(* IEC 61131-3 sources: SmartHomeNew/snapshots/2026-05-25 (part 6) *)

(* ---- PRG_Policy.st ---- *)
PROGRAM PRG_Policy
VAR
    L_Away_Elapsed_MS : UDINT;
    L_Restore_Elapsed_MS : UDINT;
    L_Return_Delta_MS : UDINT;
    L_Return_Grace_Elapsed_MS : UDINT;
    L_Security_Boost_Elapsed_MS : UDINT;
    L_Entrance_Assist_Elapsed_MS : UDINT;
    L_Away_Return_Window_Reached : BOOL;
    L_Entrance_Door_Open : BOOL;
    L_Entrance_Dark_Active : BOOL;
    L_Entrance_Motion_Active : BOOL;
    L_Previous_Away_Active : BOOL := FALSE;
    L_Previous_Away_Level : BYTE := 0;
    L_Security_Alarm_Prev : BOOL := FALSE;
    L_Entrance_Door_Open_Prev : BOOL := FALSE;
END_VAR

GVL_POLICY.G_Away_Restore_Requested := FALSE;

// ============================================================
// CONFIGURATION SAFETY CLAMP
// ============================================================
// Configuration validation is diagnostic-only here.
// System mode ownership remains in FB_State_Manager via
// FB_System_Health_Orchestrator. Policy must not directly write
// GVL_STATE.G_System_Mode.
IF GVL_CONFIG_VALIDATION.G_Config_Force_Safe_Mode AND
   (NOT GVL_CONFIG_VALIDATION.G_Config_Valid) AND
   (GVL_STATE.G_System_Mode = E_System_Operating_Mode.MODE_NORMAL) THEN
    GVL_STATUS.G_Diagnostics.Subsystem_Degraded := TRUE;
    GVL_STATUS.G_System_Mode_Text := 'CONFIG DEGRADED';
END_IF;

// ============================================================
// SCENARIO POLICY OWNER
// ============================================================

// 1. Base priority resolution
IF GVL_STATE.G_System_Mode = E_System_Operating_Mode.MODE_SAFE_STOP THEN
    GVL_POLICY.G_Scenario_Intent := E_SCENARIO_TYPE.SCENARIO_NONE;
    GVL_POLICY.G_Scenario_Source := SRC_SAFETY;

ELSIF GVL_POLICY.G_Scenario_Request_Operator <> E_SCENARIO_TYPE.SCENARIO_NONE THEN
    GVL_POLICY.G_Scenario_Intent := GVL_POLICY.G_Scenario_Request_Operator;
    GVL_POLICY.G_Scenario_Source := SRC_OPERATOR;

ELSIF GVL_POLICY.G_Scenario_Request_Gateway <> E_SCENARIO_TYPE.SCENARIO_NONE THEN
    GVL_POLICY.G_Scenario_Intent := GVL_POLICY.G_Scenario_Request_Gateway;
    GVL_POLICY.G_Scenario_Source := SRC_GATEWAY;

ELSIF GVL_POLICY.G_Scenario_Request_Rule <> E_SCENARIO_TYPE.SCENARIO_NONE THEN
    GVL_POLICY.G_Scenario_Intent := GVL_POLICY.G_Scenario_Request_Rule;
    GVL_POLICY.G_Scenario_Source := SRC_RULE;

ELSE
    GVL_POLICY.G_Scenario_Intent := GVL_STATUS.G_Current_Scenario;
    GVL_POLICY.G_Scenario_Source := SRC_NONE;
END_IF;

// 2. Fail-safe clamp
CASE GVL_STATE.G_System_Mode OF
    E_System_Operating_Mode.MODE_SAFE_STOP:
        GVL_POLICY.G_Scenario_Intent := E_SCENARIO_TYPE.SCENARIO_NONE;
        GVL_POLICY.G_Scenario_Source := SRC_SAFETY;

    E_System_Operating_Mode.MODE_FREEZE_PROTECTION:
        GVL_POLICY.G_Scenario_Intent := E_SCENARIO_TYPE.SCENARIO_NONE;
        GVL_POLICY.G_Scenario_Source := SRC_POLICY;

    E_System_Operating_Mode.MODE_DEGRADED:
        CASE GVL_POLICY.G_Scenario_Intent OF
            E_SCENARIO_TYPE.SCENARIO_NONE,
            E_SCENARIO_TYPE.SCENARIO_PRESENCE,
            E_SCENARIO_TYPE.SCENARIO_AWAY,
            E_SCENARIO_TYPE.SCENARIO_SLEEP:
                ;
        ELSE
            GVL_POLICY.G_Scenario_Intent := E_SCENARIO_TYPE.SCENARIO_NONE;
            GVL_POLICY.G_Scenario_Source := SRC_POLICY;
        END_CASE;
END_CASE;

// 3. Context automation
IF GVL_STATE.G_System_Mode = E_System_Operating_Mode.MODE_NORMAL THEN
    IF GVL_ALARM.G_Security_Armed AND
       (GVL_POLICY.G_Scenario_Request_Operator = E_SCENARIO_TYPE.SCENARIO_NONE) AND
       (GVL_POLICY.G_Scenario_Request_Gateway = E_SCENARIO_TYPE.SCENARIO_NONE) AND
       (GVL_POLICY.G_Scenario_Request_Rule = E_SCENARIO_TYPE.SCENARIO_NONE) AND
       (GVL_POLICY.G_Scenario_Intent <> E_SCENARIO_TYPE.SCENARIO_AWAY) THEN
        GVL_POLICY.G_Scenario_Intent := E_SCENARIO_TYPE.SCENARIO_AWAY;
        GVL_POLICY.G_Scenario_Source := SRC_POLICY;
    END_IF;
END_IF;

// 4. Degraded adaptation
IF GVL_STATE.G_System_Mode = E_System_Operating_Mode.MODE_DEGRADED THEN
    IF (GVL_POLICY.G_Scenario_Request_Operator = E_SCENARIO_TYPE.SCENARIO_NONE) AND
       (GVL_POLICY.G_Scenario_Request_Gateway = E_SCENARIO_TYPE.SCENARIO_NONE) AND
       (GVL_POLICY.G_Scenario_Request_Rule = E_SCENARIO_TYPE.SCENARIO_NONE) THEN

        IF GVL_ALARM.G_Security_Armed THEN
            GVL_POLICY.G_Scenario_Intent := E_SCENARIO_TYPE.SCENARIO_AWAY;
            GVL_POLICY.G_Scenario_Source := SRC_POLICY;

        ELSIF GVL_POLICY.G_Scenario_Intent = E_SCENARIO_TYPE.SCENARIO_PRESENCE THEN
            GVL_POLICY.G_Scenario_Intent := E_SCENARIO_TYPE.SCENARIO_SLEEP;
            GVL_POLICY.G_Scenario_Source := SRC_POLICY;
        END_IF;
    END_IF;
END_IF;

// 5. Security alarm escalation.
// On security alarm, force long-away and publish a 5-minute lighting boost.
IF GVL_ALARM.G_Security_Alarm THEN
    GVL_POLICY.G_Scenario_Intent := E_SCENARIO_TYPE.SCENARIO_AWAY;
    GVL_POLICY.G_Scenario_Source := SRC_POLICY;
    GVL_POLICY.G_Security_Alarm_Force_Long_Away := TRUE;

    IF (NOT L_Security_Alarm_Prev) AND (NOT GVL_POLICY.G_Security_Alarm_Light_Boost_Active) THEN
        GVL_POLICY.G_Security_Alarm_Light_Boost_Active := TRUE;
        GVL_POLICY.G_Security_Alarm_Light_Boost_Start_MS := GVL_TIME_SERVICE.G_Now_MS;
    END_IF;
ELSIF NOT GVL_ALARM.G_Security_Armed THEN
    GVL_POLICY.G_Security_Alarm_Force_Long_Away := FALSE;
END_IF;

IF GVL_POLICY.G_Security_Alarm_Light_Boost_Duration_MS = 0 THEN
    GVL_POLICY.G_Security_Alarm_Light_Boost_Duration_MS := 300000;
END_IF;

IF GVL_POLICY.G_Security_Alarm_Light_Boost_Active THEN
    IF GVL_TIME_SERVICE.G_Now_MS >= GVL_POLICY.G_Security_Alarm_Light_Boost_Start_MS THEN
        L_Security_Boost_Elapsed_MS := GVL_TIME_SERVICE.G_Now_MS - GVL_POLICY.G_Security_Alarm_Light_Boost_Start_MS;
    ELSE
        L_Security_Boost_Elapsed_MS := (4294967295 - GVL_POLICY.G_Security_Alarm_Light_Boost_Start_MS) + GVL_TIME_SERVICE.G_Now_MS + 1;
    END_IF;

    IF L_Security_Boost_Elapsed_MS >= GVL_POLICY.G_Security_Alarm_Light_Boost_Duration_MS THEN
        GVL_POLICY.G_Security_Alarm_Light_Boost_Active := FALSE;
    END_IF;
END_IF;

// 6. Entrance lighting assist.
// Trigger: entrance door rising edge while dark by configured source.
L_Entrance_Door_Open := FALSE;
IF (GVL_CONFIG.G_Entrance_Door_1_Index >= 1) AND (GVL_CONFIG.G_Entrance_Door_1_Index <= GVL_CONSTANTS.C_MAX_DOOR_SENSORS) THEN
    L_Entrance_Door_Open := L_Entrance_Door_Open OR GVL_STATE.G_Door_Sensors[GVL_CONFIG.G_Entrance_Door_1_Index];
END_IF;
IF (GVL_CONFIG.G_Entrance_Door_2_Index >= 1) AND (GVL_CONFIG.G_Entrance_Door_2_Index <= GVL_CONSTANTS.C_MAX_DOOR_SENSORS) THEN
    L_Entrance_Door_Open := L_Entrance_Door_Open OR GVL_STATE.G_Door_Sensors[GVL_CONFIG.G_Entrance_Door_2_Index];
END_IF;

L_Entrance_Dark_Active := FALSE;
IF GVL_CONFIG.G_Entrance_Light_Assist_Fallback_To_Night THEN
    L_Entrance_Dark_Active := GVL_STATUS.G_Is_Night;
END_IF;
IF GVL_CONFIG.G_Entrance_Light_Assist_Use_Lux_Sensor AND GVL_STATE.G_Ambient_Lux_Valid THEN
    L_Entrance_Dark_Active := L_Entrance_Dark_Active OR (GVL_STATE.G_Ambient_Lux < GVL_CONFIG.G_Entrance_Light_Assist_Lux_Threshold);
END_IF;
GVL_POLICY.G_Entrance_Light_Assist_Dark_Active := L_Entrance_Dark_Active;

IF GVL_CONFIG.G_Entrance_Light_Assist_Duration_MS = 0 THEN
    GVL_CONFIG.G_Entrance_Light_Assist_Duration_MS := 300000;
END_IF;

IF GVL_CONFIG.G_Entrance_Light_Assist_Enabled AND
   L_Entrance_Door_Open AND (NOT L_Entrance_Door_Open_Prev) AND
   L_Entrance_Dark_Active THEN
    GVL_POLICY.G_Entrance_Light_Assist_Active := TRUE;
    GVL_POLICY.G_Entrance_Light_Assist_Start_MS := GVL_TIME_SERVICE.G_Now_MS;
END_IF;

L_Entrance_Motion_Active := FALSE;
IF (GVL_CONFIG.G_Entrance_Corridor_Light_Zone >= 1) AND (GVL_CONFIG.G_Entrance_Corridor_Light_Zone <= GVL_CONSTANTS.C_MAX_LIGHT_ZONES) THEN
    L_Entrance_Motion_Active := L_Entrance_Motion_Active OR GVL_STATE.G_Motion_Sensors[GVL_CONFIG.G_Entrance_Corridor_Light_Zone];
END_IF;
IF (GVL_CONFIG.G_Entrance_Stairs_Light_Zone >= 1) AND (GVL_CONFIG.G_Entrance_Stairs_Light_Zone <= GVL_CONSTANTS.C_MAX_LIGHT_ZONES) THEN
    L_Entrance_Motion_Active := L_Entrance_Motion_Active OR GVL_STATE.G_Motion_Sensors[GVL_CONFIG.G_Entrance_Stairs_Light_Zone];
END_IF;

IF GVL_POLICY.G_Entrance_Light_Assist_Active THEN
    IF L_Entrance_Motion_Active THEN
        GVL_POLICY.G_Entrance_Light_Assist_Start_MS := GVL_TIME_SERVICE.G_Now_MS;
    END_IF;

    IF GVL_TIME_SERVICE.G_Now_MS >= GVL_POLICY.G_Entrance_Light_Assist_Start_MS THEN
        L_Entrance_Assist_Elapsed_MS := GVL_TIME_SERVICE.G_Now_MS - GVL_POLICY.G_Entrance_Light_Assist_Start_MS;
    ELSE
        L_Entrance_Assist_Elapsed_MS := (4294967295 - GVL_POLICY.G_Entrance_Light_Assist_Start_MS) + GVL_TIME_SERVICE.G_Now_MS + 1;
    END_IF;

    IF L_Entrance_Assist_Elapsed_MS >= GVL_CONFIG.G_Entrance_Light_Assist_Duration_MS THEN
        GVL_POLICY.G_Entrance_Light_Assist_Active := FALSE;
    END_IF;
END_IF;

// ============================================================
// AWAY LEVEL POLICY
// ============================================================
// 0=none, 1=short, 2=medium, 3=long.
// Short: light 100%, heating -1C, simulation off.
// Medium: light/simulation medium, heating -3C, simulation 0.3.
// Long: minimal reasonable heating economy; planned-return preheat may
// temporarily raise selected rooms before the expected arrival.
L_Away_Return_Window_Reached := FALSE;

IF GVL_POLICY.G_Scenario_Intent = E_SCENARIO_TYPE.SCENARIO_AWAY THEN
    IF NOT GVL_POLICY.G_Away_Active THEN
        GVL_POLICY.G_Away_Active := TRUE;
        GVL_POLICY.G_Away_Start_MS := GVL_TIME_SERVICE.G_Now_MS;
        GVL_POLICY.G_Away_Elapsed_MS := 0;
        GVL_POLICY.G_Away_Level := 1;
        GVL_POLICY.G_Away_Return_Preheat_Active := FALSE;
        GVL_POLICY.G_Away_Return_Grace_Active := FALSE;
        GVL_POLICY.G_Away_Return_Expired := FALSE;
    ELSE
        IF GVL_TIME_SERVICE.G_Now_MS >= GVL_POLICY.G_Away_Start_MS THEN
            L_Away_Elapsed_MS := GVL_TIME_SERVICE.G_Now_MS - GVL_POLICY.G_Away_Start_MS;
        ELSE
            L_Away_Elapsed_MS := (4294967295 - GVL_POLICY.G_Away_Start_MS) + GVL_TIME_SERVICE.G_Now_MS + 1;
        END_IF;

        GVL_POLICY.G_Away_Elapsed_MS := L_Away_Elapsed_MS;

        IF L_Away_Elapsed_MS >= GVL_POLICY.G_Away_Medium_To_Long_MS THEN
            GVL_POLICY.G_Away_Level := 3;
        ELSIF L_Away_Elapsed_MS >= GVL_POLICY.G_Away_Short_To_Medium_MS THEN
            GVL_POLICY.G_Away_Level := 2;
        ELSE
            GVL_POLICY.G_Away_Level := 1;
        END_IF;
    END_IF;

    // Planned return preheat window.
    IF GVL_POLICY.G_Away_Planned_Return_Enabled AND NOT GVL_POLICY.G_Away_Return_Expired THEN
        IF GVL_POLICY.G_Away_Planned_Return_MS >= GVL_TIME_SERVICE.G_Now_MS THEN
            L_Return_Delta_MS := GVL_POLICY.G_Away_Planned_Return_MS - GVL_TIME_SERVICE.G_Now_MS;
            L_Away_Return_Window_Reached := (L_Return_Delta_MS <= GVL_POLICY.G_Away_Preheat_Lead_MS);
        ELSE
            L_Away_Return_Window_Reached := TRUE;
        END_IF;

        IF L_Away_Return_Window_Reached THEN
            GVL_POLICY.G_Away_Return_Preheat_Active := TRUE;

            IF NOT GVL_POLICY.G_Away_Return_Grace_Active THEN
                GVL_POLICY.G_Away_Return_Grace_Active := TRUE;
                GVL_POLICY.G_Away_Return_Grace_Start_MS := GVL_TIME_SERVICE.G_Now_MS;
            END_IF;
        END_IF;

        IF GVL_POLICY.G_Away_Return_Grace_Active THEN
            IF GVL_TIME_SERVICE.G_Now_MS >= GVL_POLICY.G_Away_Return_Grace_Start_MS THEN
                L_Return_Grace_Elapsed_MS := GVL_TIME_SERVICE.G_Now_MS - GVL_POLICY.G_Away_Return_Grace_Start_MS;
            ELSE
                L_Return_Grace_Elapsed_MS := (4294967295 - GVL_POLICY.G_Away_Return_Grace_Start_MS) + GVL_TIME_SERVICE.G_Now_MS + 1;
            END_IF;

            IF L_Return_Grace_Elapsed_MS >= GVL_POLICY.G_Away_Return_Grace_MS THEN
                GVL_POLICY.G_Away_Return_Expired := TRUE;
                GVL_POLICY.G_Away_Return_Preheat_Active := FALSE;
                GVL_POLICY.G_Away_Return_Grace_Active := FALSE;
            END_IF;
        END_IF;
    ELSE
        GVL_POLICY.G_Away_Return_Preheat_Active := FALSE;
        GVL_POLICY.G_Away_Return_Grace_Active := FALSE;
    END_IF;

    IF GVL_POLICY.G_Security_Alarm_Force_Long_Away THEN
        GVL_POLICY.G_Away_Active := TRUE;
        GVL_POLICY.G_Away_Level := 3;
        GVL_POLICY.G_Away_Elapsed_MS := GVL_POLICY.G_Away_Medium_To_Long_MS;
        GVL_POLICY.G_Away_Return_Preheat_Active := FALSE;
        GVL_POLICY.G_Away_Return_Grace_Active := FALSE;
    END_IF;

    CASE GVL_POLICY.G_Away_Level OF
        1:
            GVL_POLICY.G_Away_Simulation_Active := FALSE;
            GVL_POLICY.G_Away_Simulation_Intensity := 0.0;
            GVL_POLICY.G_Away_Heating_Offset_C := -1.0;
        2:
            GVL_POLICY.G_Away_Simulation_Active := TRUE;
            GVL_POLICY.G_Away_Simulation_Intensity := 0.3;
            GVL_POLICY.G_Away_Heating_Offset_C := -3.0;
        3:
            GVL_POLICY.G_Away_Simulation_Active := TRUE;
            GVL_POLICY.G_Away_Simulation_Intensity := 0.2;

            IF GVL_POLICY.G_Away_Return_Preheat_Active THEN
                GVL_POLICY.G_Away_Heating_Offset_C := 0.0;
            ELSE
                GVL_POLICY.G_Away_Heating_Offset_C := GVL_POLICY.G_Away_Long_Economy_Setpoint_C - 22.0;
            END_IF;
    ELSE
            GVL_POLICY.G_Away_Simulation_Active := FALSE;
            GVL_POLICY.G_Away_Simulation_Intensity := 0.0;
            GVL_POLICY.G_Away_Heating_Offset_C := 0.0;
    END_CASE;

ELSE
    IF GVL_POLICY.G_Away_Active AND (GVL_POLICY.G_Away_Level = 1) THEN
        GVL_POLICY.G_Away_Restore_Requested := TRUE;
        GVL_POLICY.G_Away_Restore_Active := TRUE;
        GVL_POLICY.G_Away_Restore_Start_MS := GVL_TIME_SERVICE.G_Now_MS;
    END_IF;

    GVL_POLICY.G_Away_Active := FALSE;
    GVL_POLICY.G_Away_Level := 0;
    GVL_POLICY.G_Away_Elapsed_MS := 0;
    GVL_POLICY.G_Away_Simulation_Active := FALSE;
    GVL_POLICY.G_Away_Simulation_Intensity := 0.0;
    GVL_POLICY.G_Away_Heating_Offset_C := 0.0;
    GVL_POLICY.G_Away_Return_Preheat_Active := FALSE;
    GVL_POLICY.G_Away_Return_Grace_Active := FALSE;
    GVL_POLICY.G_Away_Return_Expired := FALSE;
END_IF;

IF GVL_POLICY.G_Away_Restore_Active THEN
    IF GVL_TIME_SERVICE.G_Now_MS >= GVL_POLICY.G_Away_Restore_Start_MS THEN
        L_Restore_Elapsed_MS := GVL_TIME_SERVICE.G_Now_MS - GVL_POLICY.G_Away_Restore_Start_MS;
    ELSE
        L_Restore_Elapsed_MS := (4294967295 - GVL_POLICY.G_Away_Restore_Start_MS) + GVL_TIME_SERVICE.G_Now_MS + 1;
    END_IF;

    IF L_Restore_Elapsed_MS >= GVL_POLICY.G_Away_Restore_Duration_MS THEN
        GVL_POLICY.G_Away_Restore_Progress := 1.0;
        GVL_POLICY.G_Away_Restore_Active := FALSE;
    ELSE
        GVL_POLICY.G_Away_Restore_Progress := TO_REAL(L_Restore_Elapsed_MS) / TO_REAL(GVL_POLICY.G_Away_Restore_Duration_MS);
    END_IF;
ELSE
    GVL_POLICY.G_Away_Restore_Progress := 0.0;
END_IF;

L_Previous_Away_Active := GVL_POLICY.G_Away_Active;
L_Previous_Away_Level := GVL_POLICY.G_Away_Level;
L_Security_Alarm_Prev := GVL_ALARM.G_Security_Alarm;
L_Entrance_Door_Open_Prev := L_Entrance_Door_Open;

// 5. Heating bridge
// Policy publishes preheat intent only. Actual per-circuit comfort/economy
// target selection is owned by FB_Heating_Circuit_Control through
// ST_FloorHeating_Circuit_Config.
GVL_STATE.G_Preheat_Request :=
    GVL_POLICY.G_Rule_Preheat_Request OR GVL_POLICY.G_Away_Return_Preheat_Active;
GVL_HEATING_REQUEST.G_Preheat_Request := GVL_STATE.G_Preheat_Request;
GVL_HEATING_REQUEST.G_Target_Temperature := GVL_STATE.G_Target_Temperature;

GVL_STATE.G_Freeze_Request :=
    (GVL_STATE.G_System_Mode = E_System_Operating_Mode.MODE_FREEZE_PROTECTION);
GVL_HEATING_REQUEST.G_Freeze_Request := GVL_STATE.G_Freeze_Request;

PRG_Away_Restore_Manager();
END_PROGRAM

(* ---- PRG_PreOutput_Safety_Barrier.st ---- *)
PROGRAM PRG_PreOutput_Safety_Barrier
VAR
    L_i : INT;
    L_Now_MS : UDINT;
    L_Block_IO : BOOL := FALSE;
    L_Error_Code : UDINT := 0;
    L_Error_Text : STRING(160) := '';
    L_Any_Manifold_Pump_On : BOOL := FALSE;
    L_Prev_Block_IO : BOOL;

    L_Selective_Projection_Active : BOOL;
    L_Global_Fallback_Active : BOOL;
    L_Runtime_Projection_Healthy : BOOL;

    L_Finalized_Publication_Continuity : BOOL;
    L_Physical_Causality_Healthy : BOOL;
    L_Command_Telemetry_Epoch_Aligned : BOOL;
    L_Physical_Ack_Fresh : BOOL;

    fbLog : FB_LogEvent;
END_VAR

L_Now_MS := GVL_STATUS.G_System_Time_MS;
L_Block_IO := FALSE;
L_Error_Code := 0;
L_Error_Text := '';
L_Any_Manifold_Pump_On := FALSE;
L_Prev_Block_IO := GVL_COMMAND_VERIFY.PreOutput_Block_IO;

L_Selective_Projection_Active :=
    GVL_Water_Isolation_Authority.G_Any_Selective_Authority_Allowed;

L_Global_Fallback_Active :=
    GVL_Water_Isolation_Authority.G_Any_Global_Fallback_Required;

L_Runtime_Projection_Healthy :=
    GVL_Water_Output_Reconciliation.G_Runtime_Valid
    AND NOT GVL_Water_Output_Reconciliation.G_Any_Conflict_Detected;

// Command shadow is now the command ownership surface for domain execution.
// Legacy GVL_COMMAND mismatch must not block physical publication.
GVL_COMMAND_VERIFY.Command_Match_OK := TRUE;
GVL_COMMAND_VERIFY.Command_Mismatch_Active := FALSE;
GVL_COMMAND_VERIFY.Command_Mismatch_Count := 0;

// Command ↔ telemetry epoch binding.
L_Command_Telemetry_Epoch_Aligned :=
    GVL_TELEMETRY.Command_Epoch = GVL_OUTPUT_EPOCH.Output_Publication_Epoch
    AND GVL_TELEMETRY.Telemetry_Epoch = GVL_OUTPUT_EPOCH.Output_Publication_Epoch
    AND GVL_TELEMETRY.Telemetry_Epoch >=
        GVL_TELEMETRY.Last_Acknowledged_Command_Epoch;

// Physical acknowledgment freshness.
L_Physical_Ack_Fresh :=
    (L_Now_MS - GVL_TELEMETRY.Last_Physical_Ack_Time_MS) <= 5000;

// Physical causality evidence.
L_Physical_Causality_Healthy :=
    GVL_TELEMETRY.Telemetry_Runtime_Valid
    AND GVL_TELEMETRY.Telemetry_Freshness_Valid
    AND NOT GVL_TELEMETRY.Telemetry_Lease_Expired
    AND NOT GVL_TELEMETRY.Telemetry_Quarantine_Active
    AND GVL_TELEMETRY.Command_Telemetry_Causality_Valid
    AND NOT GVL_TELEMETRY.Command_Telemetry_Divergence_Detected
    AND GVL_TELEMETRY.Actuator_Feedback_Valid
    AND GVL_TELEMETRY.Actuator_Feedback_Fresh
    AND GVL_TELEMETRY.Physical_Effect_Confirmed
    AND L_Command_Telemetry_Epoch_Aligned
    AND L_Physical_Ack_Fresh
    AND NOT GVL_TELEMETRY.Telemetry_Replay_Suspected;

// Finalized publication continuity proof chain.
L_Finalized_Publication_Continuity :=
    GVL_SEMANTIC_PROGRESS.Semantic_Forward_Progress_Valid
    AND GVL_SEMANTIC_PROGRESS.Semantic_Execution_Continuity_OK
    AND NOT GVL_SEMANTIC_PROGRESS.Semantic_Stagnation_Detected
    AND NOT GVL_SEMANTIC_PROGRESS.Semantic_Replay_Suspected
    AND NOT GVL_SEMANTIC_PROGRESS.Semantic_Livelock_Suspected
    AND NOT GVL_SEMANTIC_PROGRESS.Semantic_Deadlock_Suspected
    AND NOT GVL_SEMANTIC_PROGRESS.Semantic_Progress_Lease_Expired
    AND NOT GVL_SEMANTIC_PROGRESS.Semantic_Progress_Quarantine_Active
    AND GVL_RUNTIME_SNAPSHOT.Snapshot_Frozen
    AND GVL_RUNTIME_SNAPSHOT.Snapshot_Publication_Allowed
    AND GVL_RUNTIME_SNAPSHOT.Snapshot_Copy_Valid
    AND GVL_RUNTIME_SNAPSHOT.Snapshot_Isolation_Valid
    AND NOT GVL_RUNTIME_SNAPSHOT.Snapshot_Mutation_Detected
    AND GVL_DISTRIBUTED_SNAPSHOT.Distributed_Publication_Reconciled
    AND GVL_DISTRIBUTED_SNAPSHOT.Distributed_Publication_Freeze_Valid
    AND GVL_DISTRIBUTED_SNAPSHOT.Distributed_Snapshot_Consistent
    AND GVL_DISTRIBUTED_COMMIT.Distributed_Commit_Valid
    AND GVL_DISTRIBUTED_COMMIT.Publication_Prepare_Valid
    AND GVL_DISTRIBUTED_COMMIT.Publication_Commit_Confirmed
    AND NOT GVL_DISTRIBUTED_COMMIT.Peer_Commit_Mismatch
    AND NOT GVL_DISTRIBUTED_COMMIT.Distributed_Commit_Quarantine_Active
    AND NOT GVL_DISTRIBUTED_COMMIT.Commit_Lease_Expired
    AND GVL_OUTPUT_EPOCH.Output_Publication_Valid
    AND GVL_OUTPUT_EPOCH.Output_Runtime_Epoch_Valid
    AND NOT GVL_OUTPUT_EPOCH.Output_Lease_Expired
    AND NOT GVL_OUTPUT_EPOCH.Output_Forced_Safe_Decay;

IF (NOT L_Block_IO)
   AND (NOT L_Finalized_Publication_Continuity) THEN
    L_Block_IO := TRUE;
    L_Error_Code := 3999;
    L_Error_Text := 'PreOutput finalized publication continuity invalid';
END_IF;

IF (NOT L_Block_IO)
   AND (NOT L_Physical_Causality_Healthy) THEN
    L_Block_IO := TRUE;
    L_Error_Code := 3998;
    L_Error_Text := 'Physical causality evidence invalid';
END_IF;

IF (NOT L_Block_IO) AND (NOT GVL_STATUS.G_Is_Active_PLC) THEN
    L_Block_IO := TRUE;
    L_Error_Code := 4000;
    L_Error_Text := 'PreOutput inactive PLC';
END_IF;

GVL_COMMAND_VERIFY.PreOutput_Physical_Causality_Valid :=
    L_Physical_Causality_Healthy;

GVL_COMMAND_VERIFY.PreOutput_Barrier_OK := NOT L_Block_IO;
GVL_COMMAND_VERIFY.PreOutput_Block_IO := L_Block_IO;
GVL_COMMAND_VERIFY.PreOutput_Last_Error_Code := L_Error_Code;
GVL_COMMAND_VERIFY.PreOutput_Last_Error_Text := L_Error_Text;

IF L_Block_IO THEN
    GVL_COMMAND_VERIFY.PreOutput_Last_Error_Time_MS := L_Now_MS;
    IF NOT L_Prev_Block_IO THEN
        GVL_COMMAND_VERIFY.PreOutput_Block_Count :=
            GVL_COMMAND_VERIFY.PreOutput_Block_Count + 1;
        fbLog(
            VI_Event_Type := 1002,
            VI_Timestamp := L_Now_MS,
            VI_Param1 := L_Error_Code,
            VI_Param2 := GVL_COMMAND_VERIFY.PreOutput_Block_Count
        );
    END_IF;
END_IF;

END_PROGRAM

(* ---- PRG_Recovery_Domain.st ---- *)
PROGRAM PRG_Recovery_Domain
// SEMANTIC DOMAIN WRAPPER
// PRESERVES ORIGINAL EXECUTION ORDER

PRG_Recovery_Cleanup_Governor();
PRG_Deterministic_Recovery_Path_Governor();
PRG_Recovery_Ordering_Integrity_Governor();
PRG_Recovery_Reactivation_Control_Governor();
PRG_Authority_Resurrection_Boundary_Governor();

PRG_Energy_Resurrection_Boundary_Governor();
PRG_Physical_Deadlock_Resolution_Governor();

END_PROGRAM

(* ---- PRG_Recovery_Ordering_Integrity_Governor.st ---- *)
PROGRAM PRG_Recovery_Ordering_Integrity_Governor
IF GVL_DETERMINISTIC_RECOVERY_PATH_FABRIC.Deterministic_Recovery_Path_Granted
AND NOT GVL_RECOVERY_ORDERING_INTEGRITY_FABRIC.Unsafe_Recovery_Reordering_Detected
AND NOT GVL_RECOVERY_ORDERING_INTEGRITY_FABRIC.CrossDomain_Reactivation_Race
AND NOT GVL_RECOVERY_ORDERING_INTEGRITY_FABRIC.Recovery_Topology_Divergence
AND NOT GVL_RECOVERY_ORDERING_INTEGRITY_FABRIC.Residual_Unsafe_Reactivation_Detected THEN

    GVL_RECOVERY_ORDERING_INTEGRITY_FABRIC.Recovery_Ordering_Integrity_Valid := TRUE;
    GVL_RECOVERY_ORDERING_INTEGRITY_FABRIC.CrossDomain_Recovery_Ordering_Stable := TRUE;
    GVL_RECOVERY_ORDERING_INTEGRITY_FABRIC.Recovery_Authority_Sequencing_Canonical := TRUE;
    GVL_RECOVERY_ORDERING_INTEGRITY_FABRIC.Physical_Reactivation_Topology_Safe := TRUE;
END_IF;
END_PROGRAM

(* ---- PRG_Resource_Starvation_Boundary_Governor.st ---- *)
PROGRAM PRG_Resource_Starvation_Boundary_Governor
IF GVL_EXECUTION_PROGRESS_CAUSALITY_FABRIC.Execution_Progress_Causality_Granted
AND NOT GVL_RESOURCE_STARVATION_BOUNDARY_FABRIC.Resource_Starvation_Detected
AND NOT GVL_RESOURCE_STARVATION_BOUNDARY_FABRIC.Scheduler_Starvation_Detected
AND NOT GVL_RESOURCE_STARVATION_BOUNDARY_FABRIC.Distributed_Allocation_Deadlock_Detected THEN

    GVL_RESOURCE_STARVATION_BOUNDARY_FABRIC.Resource_Starvation_Boundary_Valid := TRUE;
    GVL_RESOURCE_STARVATION_BOUNDARY_FABRIC.Resource_Starvation_Boundary_Granted := TRUE;
    GVL_RESOURCE_STARVATION_BOUNDARY_FABRIC.Resource_Starvation_Bounded := TRUE;
    GVL_RESOURCE_STARVATION_BOUNDARY_FABRIC.Fair_Execution_Scheduling_Valid := TRUE;
END_IF;
END_PROGRAM

(* ---- PRG_Runtime_Assumption_Integrity_Governor.st ---- *)
PROGRAM PRG_Runtime_Assumption_Integrity_Governor
// PASSIVE ASSUMPTION OBSERVABILITY ONLY

GVL_RUNTIME_ASSUMPTION_INTEGRITY_FABRIC.Runtime_Assumption_Integrity_Observed :=
    GVL_PROOF_CONTINUITY_AUDIT_FABRIC.Proof_Continuity_Observed;

GVL_RUNTIME_ASSUMPTION_INTEGRITY_FABRIC.Runtime_Assumption_Lineage_Coherent := TRUE;
GVL_RUNTIME_ASSUMPTION_INTEGRITY_FABRIC.Runtime_Assumption_Stability_Observed := TRUE;

END_PROGRAM

(* ---- PRG_Runtime_IO_Validation.st ---- *)
PROGRAM PRG_Runtime_IO_Validation
VAR
    L_i : INT;
    L_Any_Exhaust_On : BOOL;
    L_Any_Supply_On : BOOL;
    L_Any_Heating_Output_On : BOOL;
    L_Any_Water_Zone_On : BOOL;
    L_Any_Access_Output_On : BOOL;
    L_Any_Lighting_Output_On : BOOL;
    L_Any_Socket_On : BOOL;
    L_Any_Freeze_Circulation_On : BOOL;
    L_Fire_Access_Valid : BOOL;
END_VAR

GVL_RUNTIME_IO_VALIDATION.G_Last_Update_MS := GVL_TIME_SERVICE.G_Now_MS;
GVL_RUNTIME_IO_VALIDATION.G_Validation_Executed := TRUE;
GVL_RUNTIME_IO_VALIDATION.G_Validation_Valid := TRUE;

L_Any_Exhaust_On := FALSE;
L_Any_Supply_On := FALSE;
L_Any_Heating_Output_On := FALSE;
L_Any_Water_Zone_On := FALSE;
L_Any_Access_Output_On := FALSE;
L_Any_Lighting_Output_On := FALSE;
L_Any_Socket_On := FALSE;
L_Any_Freeze_Circulation_On := FALSE;
L_Fire_Access_Valid := TRUE;

FOR L_i := 1 TO GVL_CONSTANTS.C_MAX_EXHAUST_FANS DO
    IF GVL_IO.AO_Exhaust_Fans[L_i] > 0 THEN
        L_Any_Exhaust_On := TRUE;
    END_IF;
END_FOR;

FOR L_i := 1 TO GVL_CONSTANTS.C_MAX_SUPPLY_FANS DO
    IF GVL_IO.AO_Supply_Fans[L_i] > 0 THEN
        L_Any_Supply_On := TRUE;
    END_IF;
END_FOR;

FOR L_i := 1 TO GVL_CONSTANTS.C_MAX_HEATING_CIRCUITS DO
    IF GVL_IO.DO_Zone_Valves[L_i] THEN
        L_Any_Heating_Output_On := TRUE;
    END_IF;
END_FOR;

FOR L_i := 1 TO GVL_CONSTANTS.C_MAX_MANIFOLDS DO
    IF GVL_IO.DO_Manifold_Pumps[L_i] OR (GVL_IO.AO_Manifold_Valves[L_i] > 0) THEN
        L_Any_Heating_Output_On := TRUE;
        L_Any_Freeze_Circulation_On := TRUE;
    END_IF;
END_FOR;

IF GVL_IO.DO_DHW_Heating_Pump
   OR GVL_IO.DO_DHW_Circ_Pump
   OR GVL_IO.DO_Backup_Circulation_Pump
   OR GVL_IO.DO_Electric_Heater_Enable THEN
    L_Any_Heating_Output_On := TRUE;
END_IF;

IF GVL_IO.DO_Backup_Circulation_Pump THEN
    L_Any_Freeze_Circulation_On := TRUE;
END_IF;

FOR L_i := 1 TO GVL_CONSTANTS.C_MAX_WATER_ZONES DO
    IF GVL_IO.DO_Water_Zone_Enable[L_i] THEN
        L_Any_Water_Zone_On := TRUE;
    END_IF;
END_FOR;

L_Any_Access_Output_On :=
    GVL_IO.DO_Gate_Open
    OR GVL_IO.DO_Wicket_Open
    OR GVL_IO.DO_Lock_1_Open
    OR GVL_IO.DO_Lock_1_Close
    OR GVL_IO.DO_Lock_2_Open
    OR GVL_IO.DO_Lock_2_Close;

IF GVL_COMMAND_SHADOW.G_Lock_1_Open AND NOT GVL_IO.DO_Lock_1_Open THEN
    L_Fire_Access_Valid := FALSE;
END_IF;
IF GVL_COMMAND_SHADOW.G_Lock_2_Open AND NOT GVL_IO.DO_Lock_2_Open THEN
    L_Fire_Access_Valid := FALSE;
END_IF;
IF GVL_COMMAND_SHADOW.G_Gate_Open AND NOT GVL_IO.DO_Gate_Open THEN
    L_Fire_Access_Valid := FALSE;
END_IF;
IF GVL_COMMAND_SHADOW.G_Wicket_Open AND NOT GVL_IO.DO_Wicket_Open THEN
    L_Fire_Access_Valid := FALSE;
END_IF;

FOR L_i := 1 TO GVL_CONSTANTS.C_MAX_LIGHT_ZONES DO
    IF GVL_IO.AO_Lighting_Levels[L_i] > 0 THEN
        L_Any_Lighting_Output_On := TRUE;
    END_IF;
END_FOR;

FOR L_i := 1 TO GVL_CONSTANTS.C_MAX_SOCKETS DO
    IF GVL_IO.DO_Sockets[L_i] THEN
        L_Any_Socket_On := TRUE;
    END_IF;
END_FOR;

GVL_RUNTIME_IO_VALIDATION.Fire_IO_Valid :=
    (NOT GVL_STATUS.G_Is_Active_PLC)
    OR (GVL_SAFETY_SHUTDOWN.G_Safety_Mode <> FIRE)
    OR (
        L_Any_Exhaust_On
        AND NOT L_Any_Supply_On
        AND L_Fire_Access_Valid
    );

GVL_RUNTIME_IO_VALIDATION.Gas_IO_Valid :=
    (NOT GVL_STATUS.G_Is_Active_PLC)
    OR (GVL_SAFETY_SHUTDOWN.G_Safety_Mode <> GAS)
    OR (
        GVL_IO.DO_Gas_Valve_Close
        AND (L_Any_Exhaust_On OR L_Any_Supply_On)
        AND NOT GVL_IO.DO_DHW_Heating_Pump
    );

GVL_RUNTIME_IO_VALIDATION.Leak_IO_Valid :=
    (GVL_SAFETY_SHUTDOWN.G_Safety_Mode <> WATER_LEAK)
    OR (
        GVL_IO.DO_Water_Valve_35_Close
        AND GVL_IO.DO_Water_Valve_36_Close
    );

GVL_RUNTIME_IO_VALIDATION.Global_Stop_IO_Valid :=
    (GVL_SAFETY_SHUTDOWN.G_Safety_Mode <> GLOBAL_STOP)
    OR (
        NOT L_Any_Heating_Output_On
        AND NOT L_Any_Exhaust_On
        AND NOT L_Any_Supply_On
        AND NOT L_Any_Water_Zone_On
        AND NOT L_Any_Access_Output_On
        AND NOT L_Any_Lighting_Output_On
        AND NOT L_Any_Socket_On
        AND GVL_IO.DO_Water_Valve_35_Close
        AND GVL_IO.DO_Water_Valve_36_Close
        AND GVL_IO.DO_Gas_Valve_Close
    );

GVL_RUNTIME_IO_VALIDATION.Inactive_PLC_IO_Valid :=
    GVL_STATUS.G_Is_Active_PLC
    OR (
        NOT L_Any_Heating_Output_On
        AND NOT L_Any_Exhaust_On
        AND NOT L_Any_Supply_On
        AND NOT L_Any_Water_Zone_On
        AND NOT L_Any_Access_Output_On
        AND NOT L_Any_Lighting_Output_On
        AND NOT L_Any_Socket_On
        AND GVL_IO.DO_Water_Valve_35_Close
        AND GVL_IO.DO_Water_Valve_36_Close
        AND GVL_IO.DO_Gas_Valve_Close
    );

GVL_RUNTIME_IO_VALIDATION.Freeze_IO_Valid :=
    (NOT GVL_STATUS.G_Is_Active_PLC)
    OR (NOT GVL_STATE.G_Safety_Freeze_Risk)
    OR L_Any_Freeze_Circulation_On;

GVL_RUNTIME_IO_VALIDATION.Any_IO_Invalid :=
    NOT GVL_RUNTIME_IO_VALIDATION.Fire_IO_Valid
    OR NOT GVL_RUNTIME_IO_VALIDATION.Gas_IO_Valid
    OR NOT GVL_RUNTIME_IO_VALIDATION.Leak_IO_Valid
    OR NOT GVL_RUNTIME_IO_VALIDATION.Global_Stop_IO_Valid
    OR NOT GVL_RUNTIME_IO_VALIDATION.Inactive_PLC_IO_Valid
    OR NOT GVL_RUNTIME_IO_VALIDATION.Freeze_IO_Valid;

IF GVL_RUNTIME_IO_VALIDATION.Any_IO_Invalid THEN
    GVL_RUNTIME_IO_VALIDATION.G_Validation_Valid := FALSE;
    GVL_RUNTIME_IO_VALIDATION.Status_Code := 1;
    GVL_RUNTIME_IO_VALIDATION.Status_Text := 'Runtime physical IO validation mismatch';
ELSE
    GVL_RUNTIME_IO_VALIDATION.Status_Code := 0;
    GVL_RUNTIME_IO_VALIDATION.Status_Text := 'Runtime physical IO validation nominal';
END_IF;

// >>> BULK_SYNC_ANCHOR: PRG_Runtime_IO_Validation <<<
END_PROGRAM

(* ---- PRG_Runtime_Scenario_Validation.st ---- *)
PROGRAM PRG_Runtime_Scenario_Validation
// Observational runtime scenario validator.
// Checks that domain execution policy matches current scenario/safety context.
// Does not gate execution and does not write physical outputs.

GVL_RUNTIME_SCENARIO_VALIDATION.G_Last_Update_MS := GVL_TIME_SERVICE.G_Now_MS;
GVL_RUNTIME_SCENARIO_VALIDATION.G_Validation_Executed := TRUE;
GVL_RUNTIME_SCENARIO_VALIDATION.G_Validation_Valid := TRUE;

GVL_RUNTIME_SCENARIO_VALIDATION.Security_Context_Active :=
    GVL_ALARM.G_Security_Armed
    OR GVL_ALARM.G_Security_Alarm;

GVL_RUNTIME_SCENARIO_VALIDATION.Away_Context_Active :=
    GVL_STATUS.G_Current_Scenario = SCENARIO_AWAY;

GVL_RUNTIME_SCENARIO_VALIDATION.Presence_Context_Active :=
    GVL_STATUS.G_Current_Scenario = SCENARIO_PRESENCE;

GVL_RUNTIME_SCENARIO_VALIDATION.Fire_Context_Active :=
    GVL_SAFETY_SHUTDOWN.G_Safety_Mode = FIRE;

GVL_RUNTIME_SCENARIO_VALIDATION.Gas_Context_Active :=
    GVL_SAFETY_SHUTDOWN.G_Safety_Mode = GAS;

GVL_RUNTIME_SCENARIO_VALIDATION.Leak_Context_Active :=
    GVL_SAFETY_SHUTDOWN.G_Safety_Mode = WATER_LEAK;

GVL_RUNTIME_SCENARIO_VALIDATION.Global_Stop_Context_Active :=
    GVL_SAFETY_SHUTDOWN.G_Safety_Mode = GLOBAL_STOP;

GVL_RUNTIME_SCENARIO_VALIDATION.Freeze_Context_Active :=
    GVL_STATE.G_Safety_Freeze_Risk
    OR GVL_INPUT.IN_Freeze_Request;

GVL_RUNTIME_SCENARIO_VALIDATION.Heating_Demand_Context_Active :=
    GVL_INPUT.IN_Preheat_Request
    OR GVL_INPUT.IN_Freeze_Request
    OR GVL_HEATING_OUTPUT.DO_DHW_Heating_Pump
    OR GVL_HEATING_OUTPUT.DO_DHW_Circ_Pump
    OR GVL_HEATING_OUTPUT.DO_Backup_Circulation_Pump
    OR GVL_HEATING_OUTPUT.DO_Electric_Heater_Enable;

GVL_RUNTIME_SCENARIO_VALIDATION.Vent_Boost_Context_Active :=
    GVL_INTENT_BEHAVIOR.I_Request_Ventilation_Boost
    OR GVL_COMMAND_SHADOW.G_Vent_PV3_Boost
    OR GVL_COMMAND_SHADOW.G_Exhaust_100_Req
    OR GVL_COMMAND_SHADOW.G_Vent_Smoke_Exhaust;

GVL_RUNTIME_SCENARIO_VALIDATION.Access_Command_Context_Active :=
    GVL_COMMAND_SHADOW.G_Lock_1_Open
    OR GVL_COMMAND_SHADOW.G_Lock_1_Close
    OR GVL_COMMAND_SHADOW.G_Lock_2_Open
    OR GVL_COMMAND_SHADOW.G_Lock_2_Close
    OR GVL_COMMAND_SHADOW.G_Gate_Open
    OR GVL_COMMAND_SHADOW.G_Wicket_Open
    OR GVL_ACCESS_RUNTIME.G_Any_Pulse_Active;

GVL_RUNTIME_SCENARIO_VALIDATION.Idle_Context_Active :=
    NOT GVL_RUNTIME_SCENARIO_VALIDATION.Security_Context_Active
    AND NOT GVL_RUNTIME_SCENARIO_VALIDATION.Away_Context_Active
    AND NOT GVL_RUNTIME_SCENARIO_VALIDATION.Presence_Context_Active
    AND NOT GVL_RUNTIME_SCENARIO_VALIDATION.Fire_Context_Active
    AND NOT GVL_RUNTIME_SCENARIO_VALIDATION.Gas_Context_Active
    AND NOT GVL_RUNTIME_SCENARIO_VALIDATION.Leak_Context_Active
    AND NOT GVL_RUNTIME_SCENARIO_VALIDATION.Global_Stop_Context_Active
    AND NOT GVL_RUNTIME_SCENARIO_VALIDATION.Freeze_Context_Active
    AND NOT GVL_RUNTIME_SCENARIO_VALIDATION.Heating_Demand_Context_Active
    AND NOT GVL_RUNTIME_SCENARIO_VALIDATION.Vent_Boost_Context_Active
    AND NOT GVL_RUNTIME_SCENARIO_VALIDATION.Access_Command_Context_Active;

GVL_RUNTIME_SCENARIO_VALIDATION.Idle_Context_Valid :=
    (NOT GVL_RUNTIME_SCENARIO_VALIDATION.Idle_Context_Active)
    OR (
        GVL_DOMAIN_EXECUTION_POLICY.Access_Mode = 0
        AND GVL_DOMAIN_EXECUTION_POLICY.Lighting_Mode = 0
        AND GVL_DOMAIN_EXECUTION_POLICY.Water_Mode = 0
        AND GVL_DOMAIN_EXECUTION_POLICY.Heating_Mode = 0
        AND GVL_DOMAIN_EXECUTION_POLICY.Vent_Mode = 0
    );

GVL_RUNTIME_SCENARIO_VALIDATION.Security_Context_Valid :=
    (NOT GVL_RUNTIME_SCENARIO_VALIDATION.Security_Context_Active)
    OR (
        GVL_DOMAIN_EXECUTION_POLICY.Access_Mode >= 1
        AND GVL_DOMAIN_EXECUTION_POLICY.Lighting_Mode >= 1
        AND GVL_DOMAIN_EXECUTION_POLICY.Water_Mode >= 1
    );

GVL_RUNTIME_SCENARIO_VALIDATION.Fire_Context_Valid :=
    (NOT GVL_RUNTIME_SCENARIO_VALIDATION.Fire_Context_Active)
    OR (
        GVL_DOMAIN_EXECUTION_POLICY.Access_Mode = 2
        AND GVL_DOMAIN_EXECUTION_POLICY.Lighting_Mode = 2
        AND GVL_DOMAIN_EXECUTION_POLICY.Vent_Mode = 2
    );

GVL_RUNTIME_SCENARIO_VALIDATION.Gas_Context_Valid :=
    (NOT GVL_RUNTIME_SCENARIO_VALIDATION.Gas_Context_Active)
    OR (
        GVL_DOMAIN_EXECUTION_POLICY.Access_Mode = 2
        AND GVL_DOMAIN_EXECUTION_POLICY.Vent_Mode = 2
        AND GVL_DOMAIN_EXECUTION_POLICY.Heating_Mode = 2
    );

GVL_RUNTIME_SCENARIO_VALIDATION.Leak_Context_Valid :=
    (NOT GVL_RUNTIME_SCENARIO_VALIDATION.Leak_Context_Active)
    OR (GVL_DOMAIN_EXECUTION_POLICY.Water_Mode = 2);

GVL_RUNTIME_SCENARIO_VALIDATION.Global_Stop_Context_Valid :=
    (NOT GVL_RUNTIME_SCENARIO_VALIDATION.Global_Stop_Context_Active)
    OR (
        GVL_DOMAIN_EXECUTION_POLICY.Heating_Mode = 2
        AND GVL_DOMAIN_EXECUTION_POLICY.Vent_Mode = 2
        AND GVL_DOMAIN_EXECUTION_POLICY.Water_Mode = 2
    );

GVL_RUNTIME_SCENARIO_VALIDATION.Freeze_Context_Valid :=
    (NOT GVL_RUNTIME_SCENARIO_VALIDATION.Freeze_Context_Active)
    OR (GVL_DOMAIN_EXECUTION_POLICY.Heating_Mode >= 1);

GVL_RUNTIME_SCENARIO_VALIDATION.Heating_Context_Valid :=
    (NOT GVL_RUNTIME_SCENARIO_VALIDATION.Heating_Demand_Context_Active)
    OR (GVL_DOMAIN_EXECUTION_POLICY.Heating_Mode >= 1);

GVL_RUNTIME_SCENARIO_VALIDATION.Vent_Context_Valid :=
    (NOT GVL_RUNTIME_SCENARIO_VALIDATION.Vent_Boost_Context_Active)
    OR (GVL_DOMAIN_EXECUTION_POLICY.Vent_Mode >= 1);

GVL_RUNTIME_SCENARIO_VALIDATION.Access_Context_Valid :=
    (NOT GVL_RUNTIME_SCENARIO_VALIDATION.Access_Command_Context_Active)
    OR (GVL_DOMAIN_EXECUTION_POLICY.Access_Mode = 2);

GVL_RUNTIME_SCENARIO_VALIDATION.Any_Context_Invalid :=
    NOT GVL_RUNTIME_SCENARIO_VALIDATION.Idle_Context_Valid
    OR NOT GVL_RUNTIME_SCENARIO_VALIDATION.Security_Context_Valid
    OR NOT GVL_RUNTIME_SCENARIO_VALIDATION.Fire_Context_Valid
    OR NOT GVL_RUNTIME_SCENARIO_VALIDATION.Gas_Context_Valid
    OR NOT GVL_RUNTIME_SCENARIO_VALIDATION.Leak_Context_Valid
    OR NOT GVL_RUNTIME_SCENARIO_VALIDATION.Global_Stop_Context_Valid
    OR NOT GVL_RUNTIME_SCENARIO_VALIDATION.Freeze_Context_Valid
    OR NOT GVL_RUNTIME_SCENARIO_VALIDATION.Heating_Context_Valid
    OR NOT GVL_RUNTIME_SCENARIO_VALIDATION.Vent_Context_Valid
    OR NOT GVL_RUNTIME_SCENARIO_VALIDATION.Access_Context_Valid;

IF GVL_RUNTIME_SCENARIO_VALIDATION.Any_Context_Invalid THEN
    GVL_RUNTIME_SCENARIO_VALIDATION.G_Validation_Valid := FALSE;
    GVL_RUNTIME_SCENARIO_VALIDATION.Status_Code := 1;
    GVL_RUNTIME_SCENARIO_VALIDATION.Status_Text := 'Runtime scenario validation mismatch';
ELSE
    GVL_RUNTIME_SCENARIO_VALIDATION.Status_Code := 0;
    GVL_RUNTIME_SCENARIO_VALIDATION.Status_Text := 'Runtime scenario validation nominal';
END_IF;

// >>> BULK_SYNC_ANCHOR: PRG_Runtime_Scenario_Validation <<<
END_PROGRAM

(* ---- PRG_Safety_Selector.st ---- *)
PROGRAM PRG_Safety_Selector
VAR
    L_i : INT;
END_VAR

GVL_Safety_Selector.G_CO_Effective := 0.0;
GVL_Safety_Selector.G_Methane_Effective := 0.0;
GVL_Safety_Selector.G_Smoke_Effective := FALSE;

FOR L_i := 1 TO GVL_CONSTANTS.C_MAX_CO_SENSORS DO
    GVL_Safety_Selector.G_CO_Effective_Array[L_i] := GVL_STATE.G_CO_Sensors[L_i];
    IF GVL_STATE.G_CO_Sensors[L_i] > GVL_Safety_Selector.G_CO_Effective THEN
        GVL_Safety_Selector.G_CO_Effective := GVL_STATE.G_CO_Sensors[L_i];
    END_IF;
END_FOR;

FOR L_i := 1 TO GVL_CONSTANTS.C_MAX_METHANE_SENSORS DO
    GVL_Safety_Selector.G_Methane_Effective_Array[L_i] := GVL_STATE.G_Methane_Sensors[L_i];
    IF GVL_STATE.G_Methane_Sensors[L_i] > GVL_Safety_Selector.G_Methane_Effective THEN
        GVL_Safety_Selector.G_Methane_Effective := GVL_STATE.G_Methane_Sensors[L_i];
    END_IF;
END_FOR;

FOR L_i := 1 TO GVL_CONSTANTS.C_MAX_SMOKE_SENSORS DO
    GVL_Safety_Selector.G_Smoke_Effective_Array[L_i] := GVL_STATE.G_Smoke_Sensors[L_i];
    GVL_Safety_Selector.G_Smoke_Effective :=
        GVL_Safety_Selector.G_Smoke_Effective
        OR GVL_STATE.G_Smoke_Sensors[L_i];
END_FOR;

// >>> BULK_SYNC_ANCHOR: PRG_Safety_Selector <<<
END_PROGRAM

(* ---- PRG_Safety_Shutdown.st ---- *)
PROGRAM PRG_Safety_Shutdown
VAR
    L_Mode : E_Safety_Mode := NORMAL;
END_VAR

// Input degraded forces safe stop first
IF GVL_INPUT.IN_Input_Degraded THEN
    L_Mode := GLOBAL_STOP;
ELSE

    // Priority: FIRE > GAS > WATER > GLOBAL_STOP > NORMAL

    IF GVL_INTENT_SAFETY.I_Fire_Alarm_Active THEN
        L_Mode := FIRE;
    ELSIF GVL_INTENT_SAFETY.I_Gas_Close_Required OR GVL_INTENT_SAFETY.I_Test_Timeout_Gas_Close THEN
        L_Mode := GAS;
    ELSIF GVL_INTENT_SAFETY.I_Water_Main_Close_Required OR GVL_INTENT_SAFETY.I_Test_Timeout_Water_Close THEN
        L_Mode := WATER_LEAK;
    ELSIF GVL_INTENT_SAFETY.I_System_Safe_Stop_Required THEN
        L_Mode := GLOBAL_STOP;
    ELSE
        L_Mode := NORMAL;
    END_IF;

END_IF;

GVL_SAFETY_SHUTDOWN.G_Safety_Mode := L_Mode;
GVL_SAFETY_SHUTDOWN.G_Safety_Active := (L_Mode <> NORMAL);

// >>> BULK_SYNC_ANCHOR: PRG_Safety_Shutdown <<<
END_PROGRAM

(* ---- PRG_Semantic_Commit_Governor.st ---- *)
PROGRAM PRG_Semantic_Commit_Governor
VAR
    L_Now_MS : UDINT;
    L_Delta_MS : UDINT;
    L_Commit_Valid : BOOL := TRUE;
    L_Error_Code : UDINT := 0;
    L_Error_Text : STRING(160) := '';
END_VAR

L_Now_MS := GVL_STATUS.G_System_Time_MS;
L_Commit_Valid := TRUE;
L_Error_Code := 0;
L_Error_Text := '';

// ======================================================
// SEMANTIC PUBLICATION COMMIT GOVERNOR
// ======================================================
// Governs semantic publication checkpoint coherence.
// Downstream/publication continuity only.
// Does not invalidate runtime barrier, PLC fencing,
// immutable snapshots, distributed commit or IO authority.
// ======================================================

GVL_SEMANTIC_COMMIT.Semantic_Checkpoint_Mismatch := FALSE;
GVL_SEMANTIC_COMMIT.Semantic_Commit_Mismatch := FALSE;
GVL_SEMANTIC_COMMIT.Semantic_Rollback_Detected := FALSE;
GVL_SEMANTIC_COMMIT.Semantic_Replay_Fenced := FALSE;
GVL_SEMANTIC_COMMIT.Semantic_Checkpoint_Missing := FALSE;
GVL_SEMANTIC_COMMIT.Semantic_Commit_Lease_Expired := FALSE;

// ------------------------------------------------------
// Semantic checkpoint epoch progression.
// ------------------------------------------------------

GVL_SEMANTIC_COMMIT.Local_Semantic_Checkpoint_Epoch :=
    GVL_SEMANTIC_COMMIT.Local_Semantic_Checkpoint_Epoch + 1;

GVL_SEMANTIC_COMMIT.Local_Semantic_Commit_Epoch :=
    GVL_SEMANTIC_COMMIT.Local_Semantic_Commit_Epoch + 1;

// ------------------------------------------------------
// Rollback/replay fencing foundation.
// ------------------------------------------------------

IF GVL_SEMANTIC_COMMIT.Peer_Semantic_Checkpoint_Epoch
< GVL_SEMANTIC_COMMIT.Local_Semantic_Checkpoint_Epoch THEN
    GVL_SEMANTIC_COMMIT.Semantic_Rollback_Detected := TRUE;
    GVL_SEMANTIC_COMMIT.Semantic_Replay_Fenced := TRUE;

    L_Commit_Valid := FALSE;
    L_Error_Code := 18000;
    L_Error_Text := 'Semantic rollback detected';
END_IF;

// ------------------------------------------------------
// Checkpoint acknowledgement foundation.
// ------------------------------------------------------

IF L_Commit_Valid THEN
    IF NOT GVL_SEMANTIC_COMMIT.Semantic_Checkpoint_Ack_Valid THEN
        GVL_SEMANTIC_COMMIT.Semantic_Checkpoint_Missing := TRUE;

        L_Commit_Valid := FALSE;
        L_Error_Code := 18001;
        L_Error_Text := 'Semantic checkpoint acknowledgement missing';
    END_IF;
END_IF;

// ------------------------------------------------------
// Semantic checkpoint mismatch foundation.
// ------------------------------------------------------

IF L_Commit_Valid THEN
    IF GVL_SEMANTIC_COMMIT.Peer_Semantic_Commit_Epoch
    <> GVL_SEMANTIC_COMMIT.Local_Semantic_Commit_Epoch THEN
        GVL_SEMANTIC_COMMIT.Semantic_Commit_Mismatch := TRUE;

        L_Commit_Valid := FALSE;
        L_Error_Code := 18002;
        L_Error_Text := 'Semantic commit mismatch detected';
    END_IF;
END_IF;

// ------------------------------------------------------
// Semantic commit lease freshness.
// ------------------------------------------------------

L_Delta_MS :=
    L_Now_MS - GVL_SEMANTIC_COMMIT.Semantic_Commit_Last_Refresh_MS;

IF L_Commit_Valid
AND GVL_SEMANTIC_COMMIT.Semantic_Commit_Lease_Active THEN
    IF L_Delta_MS > GVL_SEMANTIC_COMMIT.Semantic_Commit_Timeout_MS THEN
        GVL_SEMANTIC_COMMIT.Semantic_Commit_Lease_Expired := TRUE;

        L_Commit_Valid := FALSE;
        L_Error_Code := 18003;
        L_Error_Text := 'Semantic commit lease expired';
    END_IF;
END_IF;

// ------------------------------------------------------
// Publish semantic commit coherence foundation.
// ------------------------------------------------------

IF L_Commit_Valid THEN
    GVL_SEMANTIC_COMMIT.Semantic_Commit_Epoch :=
        GVL_SEMANTIC_COMMIT.Semantic_Commit_Epoch + 1;

    GVL_SEMANTIC_COMMIT.Semantic_Checkpoint_Epoch :=
        GVL_SEMANTIC_COMMIT.Semantic_Checkpoint_Epoch + 1;

    GVL_SEMANTIC_COMMIT.Semantic_Publication_Commit_Epoch :=
        GVL_SEMANTIC_COMMIT.Semantic_Publication_Commit_Epoch + 1;

    GVL_SEMANTIC_COMMIT.Semantic_Commit_Valid := TRUE;
    GVL_SEMANTIC_COMMIT.Semantic_Commit_Lease_Active := TRUE;
    GVL_SEMANTIC_COMMIT.Semantic_Commit_Lease_Expired := FALSE;

    GVL_SEMANTIC_COMMIT.Semantic_Commit_Quarantine_Active := FALSE;
    GVL_SEMANTIC_COMMIT.Semantic_Commit_Forced_Safe_Mode := FALSE;

    GVL_SEMANTIC_COMMIT.Semantic_Commit_Last_Refresh_MS := L_Now_MS;

    GVL_SEMANTIC_COMMIT.Semantic_Commit_Last_Error_Code := 0;
    GVL_SEMANTIC_COMMIT.Semantic_Commit_Last_Error_Text := '';
ELSE
    GVL_SEMANTIC_COMMIT.Semantic_Commit_Valid := FALSE;
    GVL_SEMANTIC_COMMIT.Semantic_Commit_Quarantine_Active := TRUE;
    GVL_SEMANTIC_COMMIT.Semantic_Commit_Forced_Safe_Mode := TRUE;

    GVL_SEMANTIC_COMMIT.Semantic_Commit_Last_Error_Code := L_Error_Code;
    GVL_SEMANTIC_COMMIT.Semantic_Commit_Last_Error_Text := L_Error_Text;

    GVL_SEMANTIC_COMMIT.Semantic_Commit_Invalidation_Count :=
        GVL_SEMANTIC_COMMIT.Semantic_Commit_Invalidation_Count + 1;
END_IF;
END_PROGRAM

(* ---- PRG_Semantic_Epoch_Invariance_Governor.st ---- *)
PROGRAM PRG_Semantic_Epoch_Invariance_Governor
VAR
    L_Now_MS : UDINT;
    L_Invariance_Valid : BOOL := TRUE;
    L_Error_Code : UDINT := 0;
    L_Error_Text : STRING(160) := '';
END_VAR

L_Now_MS := GVL_STATUS.G_System_Time_MS;
L_Invariance_Valid := TRUE;
L_Error_Code := 0;
L_Error_Text := '';

// Fail-safe defaults.
GVL_SEMANTIC_EPOCH_INVARIANCE_FABRIC.Semantic_Epoch_Invariance_Valid := FALSE;
GVL_SEMANTIC_EPOCH_INVARIANCE_FABRIC.Semantic_Epoch_Invariance_Granted := FALSE;
GVL_SEMANTIC_EPOCH_INVARIANCE_FABRIC.Semantic_Epoch_Invariance_Quarantine_Active := TRUE;

GVL_SEMANTIC_EPOCH_INVARIANCE_FABRIC.Authority_Semantics_Invariant := FALSE;
GVL_SEMANTIC_EPOCH_INVARIANCE_FABRIC.CrossEpoch_Permission_Mapping_Stable := FALSE;
GVL_SEMANTIC_EPOCH_INVARIANCE_FABRIC.Semantic_Intent_Continuity_Valid := FALSE;
GVL_SEMANTIC_EPOCH_INVARIANCE_FABRIC.Governance_Meaning_Preservation_Coherent := FALSE;
GVL_SEMANTIC_EPOCH_INVARIANCE_FABRIC.Semantic_Evolution_Lineage_Traceable := FALSE;

// Trust epoch monotonicity required.
IF NOT GVL_TRUST_EPOCH_MONOTONICITY_FABRIC.Trust_Epoch_Monotonicity_Granted THEN
    L_Invariance_Valid := FALSE;
    L_Error_Code := 49000;
    L_Error_Text := 'Trust epoch monotonicity not granted';
END_IF;

// Semantic epoch drift detectors.
IF GVL_SEMANTIC_EPOCH_INVARIANCE_FABRIC.Semantic_Authority_Drift_Detected THEN
    L_Invariance_Valid := FALSE;
    L_Error_Code := 49001;
    L_Error_Text := 'Semantic authority drift detected';
END_IF;

IF GVL_SEMANTIC_EPOCH_INVARIANCE_FABRIC.CrossEpoch_Permission_Reinterpretation THEN
    L_Invariance_Valid := FALSE;
    L_Error_Code := 49002;
    L_Error_Text := 'Cross-epoch permission reinterpretation detected';
END_IF;

IF GVL_SEMANTIC_EPOCH_INVARIANCE_FABRIC.Intent_To_Authority_Mismatch_Detected THEN
    L_Invariance_Valid := FALSE;
    L_Error_Code := 49003;
    L_Error_Text := 'Intent-to-authority mismatch detected';
END_IF;

IF GVL_SEMANTIC_EPOCH_INVARIANCE_FABRIC.Governance_Semantic_Fork_Detected THEN
    L_Invariance_Valid := FALSE;
    L_Error_Code := 49004;
    L_Error_Text := 'Governance semantic fork detected';
END_IF;

IF GVL_SEMANTIC_EPOCH_INVARIANCE_FABRIC.Semantic_Migration_Lineage_Gap_Detected THEN
    L_Invariance_Valid := FALSE;
    L_Error_Code := 49005;
    L_Error_Text := 'Semantic migration lineage gap detected';
END_IF;

IF GVL_SEMANTIC_EPOCH_INVARIANCE_FABRIC.Distributed_Semantic_Divergence_Detected THEN
    L_Invariance_Valid := FALSE;
    L_Error_Code := 49006;
    L_Error_Text := 'Distributed semantic divergence detected';
END_IF;

// Semantic invariance validation.
IF L_Invariance_Valid
AND NOT GVL_SEMANTIC_EPOCH_INVARIANCE_FABRIC.Explicit_Semantic_Migration_Governed THEN
    L_Invariance_Valid := FALSE;
    L_Error_Code := 49010;
    L_Error_Text := 'Explicit semantic migration governance invalid';
END_IF;

IF L_Invariance_Valid
AND NOT GVL_SEMANTIC_EPOCH_INVARIANCE_FABRIC.CrossEpoch_Semantic_Equivalence_Valid THEN
    L_Invariance_Valid := FALSE;
    L_Error_Code := 49011;
    L_Error_Text := 'Cross-epoch semantic equivalence invalid';
END_IF;

IF L_Invariance_Valid
AND NOT GVL_SEMANTIC_EPOCH_INVARIANCE_FABRIC.Distributed_Semantic_Consensus_Stable THEN
    L_Invariance_Valid := FALSE;
    L_Error_Code := 49012;
    L_Error_Text := 'Distributed semantic consensus invalid';
END_IF;

IF L_Invariance_Valid
AND NOT GVL_SEMANTIC_EPOCH_INVARIANCE_FABRIC.Semantic_Interpretation_Integrity_Valid THEN
    L_Invariance_Valid := FALSE;
    L_Error_Code := 49013;
    L_Error_Text := 'Semantic interpretation integrity invalid';
END_IF;

IF L_Invariance_Valid THEN
    GVL_SEMANTIC_EPOCH_INVARIANCE_FABRIC.Semantic_Epoch_Invariance_Valid := TRUE;
    GVL_SEMANTIC_EPOCH_INVARIANCE_FABRIC.Semantic_Epoch_Invariance_Granted := TRUE;
    GVL_SEMANTIC_EPOCH_INVARIANCE_FABRIC.Semantic_Epoch_Invariance_Quarantine_Active := FALSE;

    GVL_SEMANTIC_EPOCH_INVARIANCE_FABRIC.Authority_Semantics_Invariant := TRUE;
    GVL_SEMANTIC_EPOCH_INVARIANCE_FABRIC.CrossEpoch_Permission_Mapping_Stable := TRUE;
    GVL_SEMANTIC_EPOCH_INVARIANCE_FABRIC.Semantic_Intent_Continuity_Valid := TRUE;
    GVL_SEMANTIC_EPOCH_INVARIANCE_FABRIC.Governance_Meaning_Preservation_Coherent := TRUE;
    GVL_SEMANTIC_EPOCH_INVARIANCE_FABRIC.Semantic_Evolution_Lineage_Traceable := TRUE;

    GVL_SEMANTIC_EPOCH_INVARIANCE_FABRIC.Semantic_Epoch_Invariance_Epoch :=
        GVL_TRUST_EPOCH_MONOTONICITY_FABRIC.Trust_Epoch_Monotonicity_Epoch;

    GVL_SEMANTIC_EPOCH_INVARIANCE_FABRIC.Semantic_Epoch_Invariance_Epoch_Coherent := TRUE;

    GVL_SEMANTIC_EPOCH_INVARIANCE_FABRIC.Semantic_Epoch_Invariance_Last_Update_MS :=
        L_Now_MS;

    GVL_SEMANTIC_EPOCH_INVARIANCE_FABRIC.Semantic_Epoch_Invariance_Lease_Expired := FALSE;

    GVL_SEMANTIC_EPOCH_INVARIANCE_FABRIC.Semantic_Epoch_Invariance_Last_Error_Code := 0;
    GVL_SEMANTIC_EPOCH_INVARIANCE_FABRIC.Semantic_Epoch_Invariance_Last_Error_Text := '';
ELSE
    GVL_SEMANTIC_EPOCH_INVARIANCE_FABRIC.Semantic_Epoch_Invariance_Valid := FALSE;
    GVL_SEMANTIC_EPOCH_INVARIANCE_FABRIC.Semantic_Epoch_Invariance_Granted := FALSE;
    GVL_SEMANTIC_EPOCH_INVARIANCE_FABRIC.Semantic_Epoch_Invariance_Quarantine_Active := TRUE;

    GVL_SEMANTIC_EPOCH_INVARIANCE_FABRIC.Semantic_Epoch_Invariance_Lease_Expired := TRUE;

    GVL_SEMANTIC_EPOCH_INVARIANCE_FABRIC.Semantic_Epoch_Invariance_Last_Error_Code :=
        L_Error_Code;

    GVL_SEMANTIC_EPOCH_INVARIANCE_FABRIC.Semantic_Epoch_Invariance_Last_Error_Text :=
        L_Error_Text;

    GVL_SEMANTIC_EPOCH_INVARIANCE_FABRIC.Semantic_Epoch_Invariance_Invalidation_Count :=
        GVL_SEMANTIC_EPOCH_INVARIANCE_FABRIC.Semantic_Epoch_Invariance_Invalidation_Count + 1;
END_IF;

END_PROGRAM

(* ---- PRG_Semantic_Preservation_Governor.st ---- *)
PROGRAM PRG_Semantic_Preservation_Governor
VAR
    L_Now_MS : UDINT;
    L_Semantic_Valid : BOOL := TRUE;
    L_Error_Code : UDINT := 0;
    L_Error_Text : STRING(160) := '';
END_VAR

L_Now_MS := GVL_STATUS.G_System_Time_MS;
L_Semantic_Valid := TRUE;
L_Error_Code := 0;
L_Error_Text := '';

// Fail-safe defaults.
GVL_SEMANTIC_PRESERVATION_FABRIC.Semantic_Preservation_Valid := FALSE;
GVL_SEMANTIC_PRESERVATION_FABRIC.Semantic_Preservation_Granted := FALSE;
GVL_SEMANTIC_PRESERVATION_FABRIC.Semantic_Preservation_Quarantine_Active := TRUE;

GVL_SEMANTIC_PRESERVATION_FABRIC.Declared_System_Intent_Coherent := FALSE;
GVL_SEMANTIC_PRESERVATION_FABRIC.Adaptive_Policy_Bounded := FALSE;
GVL_SEMANTIC_PRESERVATION_FABRIC.Cross_Domain_Intent_Aligned := FALSE;
GVL_SEMANTIC_PRESERVATION_FABRIC.Optimization_Goals_Coherent := FALSE;
GVL_SEMANTIC_PRESERVATION_FABRIC.Behavioral_Evolution_Stable := FALSE;

// Runtime sustainability required.
IF NOT GVL_RUNTIME_SUSTAINABILITY_FABRIC.Runtime_Sustainability_Granted THEN
    L_Semantic_Valid := FALSE;
    L_Error_Code := 39000;
    L_Error_Text := 'Runtime sustainability authority not granted';
END_IF;

// Semantic drift detectors.
IF GVL_SEMANTIC_PRESERVATION_FABRIC.Adaptive_Policy_Drift_Detected THEN
    L_Semantic_Valid := FALSE;
    L_Error_Code := 39001;
    L_Error_Text := 'Adaptive policy drift detected';
END_IF;

IF GVL_SEMANTIC_PRESERVATION_FABRIC.Optimization_Semantic_Erosion_Detected THEN
    L_Semantic_Valid := FALSE;
    L_Error_Code := 39002;
    L_Error_Text := 'Optimization semantic erosion detected';
END_IF;

IF GVL_SEMANTIC_PRESERVATION_FABRIC.CrossDomain_Intent_Divergence_Detected THEN
    L_Semantic_Valid := FALSE;
    L_Error_Code := 39003;
    L_Error_Text := 'Cross-domain intent divergence detected';
END_IF;

IF GVL_SEMANTIC_PRESERVATION_FABRIC.LongTerm_Objective_Mutation_Detected THEN
    L_Semantic_Valid := FALSE;
    L_Error_Code := 39004;
    L_Error_Text := 'Long-term objective mutation detected';
END_IF;

IF GVL_SEMANTIC_PRESERVATION_FABRIC.Behavior_Learning_Instability_Detected THEN
    L_Semantic_Valid := FALSE;
    L_Error_Code := 39005;
    L_Error_Text := 'Behavior learning instability detected';
END_IF;

IF GVL_SEMANTIC_PRESERVATION_FABRIC.Silent_Governance_Reinterpretation_Detected THEN
    L_Semantic_Valid := FALSE;
    L_Error_Code := 39006;
    L_Error_Text := 'Silent governance reinterpretation detected';
END_IF;

// Immutable semantic intent validation.
IF L_Semantic_Valid
AND NOT GVL_SEMANTIC_PRESERVATION_FABRIC.Objective_Boundaries_Immutable THEN
    L_Semantic_Valid := FALSE;
    L_Error_Code := 39010;
    L_Error_Text := 'Objective boundaries immutability invalid';
END_IF;

IF L_Semantic_Valid
AND NOT GVL_SEMANTIC_PRESERVATION_FABRIC.Semantic_Governance_Coherent THEN
    L_Semantic_Valid := FALSE;
    L_Error_Code := 39011;
    L_Error_Text := 'Semantic governance coherence invalid';
END_IF;

IF L_Semantic_Valid
AND NOT GVL_SEMANTIC_PRESERVATION_FABRIC.Adaptive_Runtime_Intent_Stable THEN
    L_Semantic_Valid := FALSE;
    L_Error_Code := 39012;
    L_Error_Text := 'Adaptive runtime intent unstable';
END_IF;

IF L_Semantic_Valid
AND NOT GVL_SEMANTIC_PRESERVATION_FABRIC.LongTerm_Semantic_Evolution_Valid THEN
    L_Semantic_Valid := FALSE;
    L_Error_Code := 39013;
    L_Error_Text := 'Long-term semantic evolution invalid';
END_IF;

IF L_Semantic_Valid THEN
    GVL_SEMANTIC_PRESERVATION_FABRIC.Semantic_Preservation_Valid := TRUE;
    GVL_SEMANTIC_PRESERVATION_FABRIC.Semantic_Preservation_Granted := TRUE;
    GVL_SEMANTIC_PRESERVATION_FABRIC.Semantic_Preservation_Quarantine_Active := FALSE;

    GVL_SEMANTIC_PRESERVATION_FABRIC.Declared_System_Intent_Coherent := TRUE;
    GVL_SEMANTIC_PRESERVATION_FABRIC.Adaptive_Policy_Bounded := TRUE;
    GVL_SEMANTIC_PRESERVATION_FABRIC.Cross_Domain_Intent_Aligned := TRUE;
    GVL_SEMANTIC_PRESERVATION_FABRIC.Optimization_Goals_Coherent := TRUE;
    GVL_SEMANTIC_PRESERVATION_FABRIC.Behavioral_Evolution_Stable := TRUE;

    GVL_SEMANTIC_PRESERVATION_FABRIC.Semantic_Preservation_Epoch :=
        GVL_RUNTIME_SUSTAINABILITY_FABRIC.Runtime_Sustainability_Epoch;

    GVL_SEMANTIC_PRESERVATION_FABRIC.Semantic_Preservation_Epoch_Coherent := TRUE;

    GVL_SEMANTIC_PRESERVATION_FABRIC.Semantic_Preservation_Last_Update_MS :=
        L_Now_MS;

    GVL_SEMANTIC_PRESERVATION_FABRIC.Semantic_Preservation_Lease_Expired := FALSE;

    GVL_SEMANTIC_PRESERVATION_FABRIC.Semantic_Preservation_Last_Error_Code := 0;
    GVL_SEMANTIC_PRESERVATION_FABRIC.Semantic_Preservation_Last_Error_Text := '';
ELSE
    GVL_SEMANTIC_PRESERVATION_FABRIC.Semantic_Preservation_Valid := FALSE;
    GVL_SEMANTIC_PRESERVATION_FABRIC.Semantic_Preservation_Granted := FALSE;
    GVL_SEMANTIC_PRESERVATION_FABRIC.Semantic_Preservation_Quarantine_Active := TRUE;

    GVL_SEMANTIC_PRESERVATION_FABRIC.Semantic_Preservation_Lease_Expired := TRUE;

    GVL_SEMANTIC_PRESERVATION_FABRIC.Semantic_Preservation_Last_Error_Code :=
        L_Error_Code;

    GVL_SEMANTIC_PRESERVATION_FABRIC.Semantic_Preservation_Last_Error_Text :=
        L_Error_Text;

    GVL_SEMANTIC_PRESERVATION_FABRIC.Semantic_Preservation_Invalidation_Count :=
        GVL_SEMANTIC_PRESERVATION_FABRIC.Semantic_Preservation_Invalidation_Count + 1;
END_IF;

END_PROGRAM

(* ---- PRG_Survivability_Intelligence_Governor.st ---- *)
PROGRAM PRG_Survivability_Intelligence_Governor
// ADVISORY SURVIVABILITY INTELLIGENCE
// READ-ONLY / NON-INVASIVE
// NO ACTUATION / AUTHORITY / RECOVERY MUTATION

GVL_SURVIVABILITY_INTELLIGENCE_FABRIC.System_Survivable :=
    GVL_PHYSICAL_REALITY_VERIFICATION_FABRIC.Physical_Runtime_Reality_Valid;

GVL_SURVIVABILITY_INTELLIGENCE_FABRIC.Degraded_But_Safe :=
    GVL_RUNTIME_STATE_ALGEBRA.Current_Runtime_State = SYS_DEGRADED;

GVL_SURVIVABILITY_INTELLIGENCE_FABRIC.Isolated_But_Stable :=
    GVL_RUNTIME_STATE_ALGEBRA.Current_Runtime_State = SYS_ISOLATED;

GVL_SURVIVABILITY_INTELLIGENCE_FABRIC.Partitioned_But_Survivable :=
    GVL_RUNTIME_STATE_ALGEBRA.Current_Runtime_State = SYS_PARTITIONED;

GVL_SURVIVABILITY_INTELLIGENCE_FABRIC.Resource_Starved_But_Recoverable :=
    GVL_OPERATIONAL_INTELLIGENCE_FABRIC.Governance_Complexity_Pressure_Observed;

GVL_SURVIVABILITY_INTELLIGENCE_FABRIC.Essential_Functions_Preserved :=
    GVL_SAFETY_OBSERVABILITY_TRUTH_FABRIC.Observability_Reality_Equivalence_Granted;

IF GVL_OPERATIONAL_INTELLIGENCE_FABRIC.Governance_Saturation_Observed THEN
    GVL_SURVIVABILITY_INTELLIGENCE_FABRIC.NonEssential_Shedding_Recommended := TRUE;
    GVL_SURVIVABILITY_INTELLIGENCE_FABRIC.Heavy_Diagnostics_Defer_Recommended := TRUE;
    GVL_SURVIVABILITY_INTELLIGENCE_FABRIC.Trend_Analytics_Defer_Recommended := TRUE;
END_IF;

IF GVL_OPERATIONAL_INTELLIGENCE_FABRIC.Governance_Complexity_Pressure_Observed THEN
    GVL_SURVIVABILITY_INTELLIGENCE_FABRIC.Telemetry_Rate_Reduction_Recommended := TRUE;
END_IF;

IF GVL_RUNTIME_TRANSITION_SYSTEM.Illegal_Runtime_Transition_Observed THEN
    GVL_SURVIVABILITY_INTELLIGENCE_FABRIC.LongDuration_Degradation_Observed := TRUE;
    GVL_SURVIVABILITY_INTELLIGENCE_FABRIC.Chronic_Degradation_Risk_Increasing := TRUE;
    GVL_SURVIVABILITY_INTELLIGENCE_FABRIC.Survivability_Advisory_Available := TRUE;
    GVL_SURVIVABILITY_INTELLIGENCE_FABRIC.Survivability_Advisory_Code :=
        'survivability degraded under prolonged instability';
END_IF;

GVL_SURVIVABILITY_INTELLIGENCE_FABRIC.Governance_Saturation_Pressure_Observed :=
    GVL_OPERATIONAL_INTELLIGENCE_FABRIC.Governance_Saturation_Observed;

GVL_SURVIVABILITY_INTELLIGENCE_FABRIC.Distributed_Instability_Pressure_Observed :=
    NOT GVL_DISTRIBUTED_SAFETY_REALITY_CONSENSUS_FABRIC.Distributed_Safety_Consensus_Valid;

END_PROGRAM

(* ---- PRG_System_Diagnostics_Ext.st ---- *)
PROGRAM PRG_System_Diagnostics_Ext
VAR
    L_Error_Heating : BOOL;
    L_Error_Safety : BOOL;
    L_Error_IO : BOOL;

    L_Delta_Time : REAL;
    L_Now : UDINT;
    L_Last : UDINT;

    // cycle stats
    L_Cycle_MS : UDINT;
    L_Prev_Overrun : BOOL;
    L_Prev_Critical : BOOL;
    L_Prev_Error_Heating : BOOL;
    L_Prev_Error_Safety : BOOL;
    L_Prev_Error_IO : BOOL;
    fbLog : FB_LogEvent;
END_VAR

L_Now := GVL_TIME_SERVICE.G_Now_MS;
L_Last := GVL_DIAGNOSTICS_EXT.G_Last_Update_Time;

// ===============================
// CYCLE INTERVAL MEASUREMENT
// ===============================
IF L_Last = 0 THEN
    L_Cycle_MS := GVL_DIAGNOSTICS_EXT.G_Cycle_Expected_MS;
ELSE
    IF L_Now >= L_Last THEN
        L_Cycle_MS := L_Now - L_Last;
    ELSE
        L_Cycle_MS := (4294967295 - L_Last) + L_Now + 1;
    END_IF;
END_IF;

GVL_DIAGNOSTICS_EXT.G_Last_Update_Time := L_Now;
GVL_DIAGNOSTICS_EXT.G_Cycle_Last_MS := L_Cycle_MS;

// min/max
IF (GVL_DIAGNOSTICS_EXT.G_Cycle_Min_MS = 0) OR (L_Cycle_MS < GVL_DIAGNOSTICS_EXT.G_Cycle_Min_MS) THEN
    GVL_DIAGNOSTICS_EXT.G_Cycle_Min_MS := L_Cycle_MS;
END_IF;

IF L_Cycle_MS > GVL_DIAGNOSTICS_EXT.G_Cycle_Max_MS THEN
    GVL_DIAGNOSTICS_EXT.G_Cycle_Max_MS := L_Cycle_MS;
END_IF;

// average (incremental)
GVL_DIAGNOSTICS_EXT.G_Cycle_Sample_Count := GVL_DIAGNOSTICS_EXT.G_Cycle_Sample_Count + 1;
GVL_DIAGNOSTICS_EXT.G_Cycle_Avg_MS :=
    GVL_DIAGNOSTICS_EXT.G_Cycle_Avg_MS +
    (UDINT_TO_REAL(L_Cycle_MS) - GVL_DIAGNOSTICS_EXT.G_Cycle_Avg_MS) /
    UDINT_TO_REAL(GVL_DIAGNOSTICS_EXT.G_Cycle_Sample_Count);

// ===============================
// OVERRUN / CRITICAL DETECTION
// ===============================
GVL_DIAGNOSTICS_EXT.G_Cycle_Overrun_Active := (L_Cycle_MS > GVL_DIAGNOSTICS_EXT.G_Cycle_Warning_MS);
GVL_DIAGNOSTICS_EXT.G_Cycle_Critical_Active := (L_Cycle_MS > GVL_DIAGNOSTICS_EXT.G_Cycle_Critical_MS);

IF GVL_DIAGNOSTICS_EXT.G_Cycle_Overrun_Active THEN
    GVL_DIAGNOSTICS_EXT.G_Cycle_Overrun_Count := GVL_DIAGNOSTICS_EXT.G_Cycle_Overrun_Count + 1;
    GVL_DIAGNOSTICS_EXT.G_Cycle_Last_Overrun_MS := L_Cycle_MS;
    GVL_DIAGNOSTICS_EXT.G_Cycle_Last_Overrun_Time_MS := L_Now;
END_IF;

IF GVL_DIAGNOSTICS_EXT.G_Cycle_Critical_Active THEN
    GVL_DIAGNOSTICS_EXT.G_Cycle_Critical_Count := GVL_DIAGNOSTICS_EXT.G_Cycle_Critical_Count + 1;
END_IF;

// edge logging
IF GVL_DIAGNOSTICS_EXT.G_Cycle_Overrun_Active AND NOT L_Prev_Overrun THEN
    fbLog(
        VI_Event_Type := 2001,
        VI_Timestamp := L_Now,
        VI_Param1 := L_Cycle_MS,
        VI_Param2 := GVL_DIAGNOSTICS_EXT.G_Cycle_Overrun_Count
    );
END_IF;

IF GVL_DIAGNOSTICS_EXT.G_Cycle_Critical_Active AND NOT L_Prev_Critical THEN
    fbLog(
        VI_Event_Type := 2002,
        VI_Timestamp := L_Now,
        VI_Param1 := L_Cycle_MS,
        VI_Param2 := GVL_DIAGNOSTICS_EXT.G_Cycle_Critical_Count
    );
END_IF;

L_Prev_Overrun := GVL_DIAGNOSTICS_EXT.G_Cycle_Overrun_Active;
L_Prev_Critical := GVL_DIAGNOSTICS_EXT.G_Cycle_Critical_Active;

// ===============================
// EXISTING HEALTH LOGIC
// ===============================
IF L_Last = 0 THEN
    L_Delta_Time := 0.1;
ELSE
    L_Delta_Time := UDINT_TO_REAL(L_Cycle_MS) / 1000.0;
END_IF;

L_Error_Heating := GVL_STATE.G_Heating_Subsystem_Degraded;

// Extended diagnostics must use authoritative safety truth and latches,
// not stale projected GVL_STATE.G_Safety_*_Alarm compatibility fields.
L_Error_Safety :=
    GVL_HEALTH_BRIDGE.G_Gas_Detected OR
    GVL_HEALTH_BRIDGE.G_CO_Alarm_Level OR
    GVL_HEALTH_BRIDGE.G_Leak_Detected OR
    GVL_HEALTH_BRIDGE.G_Smoke_Detected OR
    GVL_STATE.G_Safety_Gas_Latched OR
    GVL_STATE.G_Safety_Leak_Latched OR
    GVL_STATE.G_Safety_Smoke_Latched;

L_Error_IO := GVL_STATE.G_Heating_IO_Fault;

IF L_Error_Heating THEN
    IF NOT L_Prev_Error_Heating THEN
        GVL_DIAGNOSTICS_EXT.G_Error_Count_Heating := GVL_DIAGNOSTICS_EXT.G_Error_Count_Heating + 1;
    END_IF;
    GVL_DIAGNOSTICS_EXT.G_Last_Error_Time_Heating := L_Now;
    GVL_DIAGNOSTICS_EXT.G_Health_Heating := GVL_DIAGNOSTICS_EXT.G_Health_Heating - (0.5 * L_Delta_Time);
ELSE
    GVL_DIAGNOSTICS_EXT.G_Health_Heating := GVL_DIAGNOSTICS_EXT.G_Health_Heating + (0.1 * L_Delta_Time);
END_IF;

IF L_Error_Safety THEN
    IF NOT L_Prev_Error_Safety THEN
        GVL_DIAGNOSTICS_EXT.G_Error_Count_Safety := GVL_DIAGNOSTICS_EXT.G_Error_Count_Safety + 1;
    END_IF;
    GVL_DIAGNOSTICS_EXT.G_Last_Error_Time_Safety := L_Now;
    GVL_DIAGNOSTICS_EXT.G_Health_Safety := GVL_DIAGNOSTICS_EXT.G_Health_Safety - (1.0 * L_Delta_Time);
ELSE
    GVL_DIAGNOSTICS_EXT.G_Health_Safety := GVL_DIAGNOSTICS_EXT.G_Health_Safety + (0.2 * L_Delta_Time);
END_IF;

IF L_Error_IO THEN
    IF NOT L_Prev_Error_IO THEN
        GVL_DIAGNOSTICS_EXT.G_Error_Count_IO := GVL_DIAGNOSTICS_EXT.G_Error_Count_IO + 1;
    END_IF;
    GVL_DIAGNOSTICS_EXT.G_Last_Error_Time_IO := L_Now;
    GVL_DIAGNOSTICS_EXT.G_Health_IO := GVL_DIAGNOSTICS_EXT.G_Health_IO - (0.5 * L_Delta_Time);
ELSE
    GVL_DIAGNOSTICS_EXT.G_Health_IO := GVL_DIAGNOSTICS_EXT.G_Health_IO + (0.1 * L_Delta_Time);
END_IF;

L_Prev_Error_Heating := L_Error_Heating;
L_Prev_Error_Safety := L_Error_Safety;
L_Prev_Error_IO := L_Error_IO;

// clamp
IF GVL_DIAGNOSTICS_EXT.G_Health_Heating < 0.0 THEN GVL_DIAGNOSTICS_EXT.G_Health_Heating := 0.0; END_IF;
IF GVL_DIAGNOSTICS_EXT.G_Health_Heating > 1.0 THEN GVL_DIAGNOSTICS_EXT.G_Health_Heating := 1.0; END_IF;

IF GVL_DIAGNOSTICS_EXT.G_Health_Safety < 0.0 THEN GVL_DIAGNOSTICS_EXT.G_Health_Safety := 0.0; END_IF;
IF GVL_DIAGNOSTICS_EXT.G_Health_Safety > 1.0 THEN GVL_DIAGNOSTICS_EXT.G_Health_Safety := 1.0; END_IF;

IF GVL_DIAGNOSTICS_EXT.G_Health_IO < 0.0 THEN GVL_DIAGNOSTICS_EXT.G_Health_IO := 0.0; END_IF;
IF GVL_DIAGNOSTICS_EXT.G_Health_IO > 1.0 THEN GVL_DIAGNOSTICS_EXT.G_Health_IO := 1.0; END_IF;

END_PROGRAM

(* ---- PRG_System_Evacuation.st ---- *)
PROGRAM PRG_System_Evacuation
VAR
    fbSystemEvacuation : FB_System_Evacuation;
END_VAR

fbSystemEvacuation();

END_PROGRAM

(* ---- PRG_System_History.st ---- *)
PROGRAM PRG_System_History
VAR
    fbHistoryManager : FB_History_Manager;
    L_History_Event : ST_History_Record;
    L_History_Write_Event : BOOL;
    L_Last_System_Mode : E_System_Operating_Mode;
    L_Last_Root_Cause : E_System_Root_Cause;
    L_Last_First_Fault_Source : INT;
    L_Last_Operator_Journal_Seq : UDINT;
    L_Last_Event_Code : UDINT;
    L_Last_Event_Value : REAL;
    L_Last_Event_Time_MS : UDINT;
END_VAR

L_History_Write_Event := FALSE;
L_History_Event.timestamp_ms := GVL_TIME_SERVICE.G_Now_MS;
L_History_Event.event_code := 0;
L_History_Event.event_value := 0.0;
L_History_Event.unit := 0;
L_History_Event.zone_id := 0;
L_History_Event.operator_id := 'SYSTEM';
L_History_Event.priority := E_ALERT_PRIORITY.ALERT_PRIORITY_HIGH;

IF GVL_STATE.G_System_Mode <> L_Last_System_Mode THEN
    L_History_Write_Event := TRUE;
    L_History_Event.event_code := 1101;
    L_History_Event.event_value := TO_REAL(TO_INT(GVL_STATE.G_System_Mode));
    L_History_Event.unit := 1;
    L_History_Event.zone_id := 0;
    L_History_Event.priority := E_ALERT_PRIORITY.ALERT_PRIORITY_HIGH;
    L_Last_System_Mode := GVL_STATE.G_System_Mode;

ELSIF GVL_SYSTEM_HEALTH.G_First_Fault_Active
      AND (GVL_SYSTEM_HEALTH.G_Root_Cause <> L_Last_Root_Cause) THEN
    L_History_Write_Event := TRUE;
    L_History_Event.event_code := 1102;
    L_History_Event.event_value := TO_REAL(TO_INT(GVL_SYSTEM_HEALTH.G_Root_Cause));
    L_History_Event.unit := 2;
    L_History_Event.zone_id := TO_BYTE(GVL_SYSTEM_HEALTH.G_First_Fault_Source);
    L_History_Event.priority := E_ALERT_PRIORITY.ALERT_PRIORITY_HIGH;
    L_Last_Root_Cause := GVL_SYSTEM_HEALTH.G_Root_Cause;

ELSIF GVL_SYSTEM_HEALTH.G_First_Fault_Active
      AND (GVL_SYSTEM_HEALTH.G_First_Fault_Source <> L_Last_First_Fault_Source) THEN
    L_History_Write_Event := TRUE;
    L_History_Event.event_code := 1103;
    L_History_Event.event_value := TO_REAL(GVL_SYSTEM_HEALTH.G_First_Fault_Source);
    L_History_Event.unit := 3;
    L_History_Event.zone_id := TO_BYTE(GVL_SYSTEM_HEALTH.G_First_Fault_Source);
    L_History_Event.priority := E_ALERT_PRIORITY.ALERT_PRIORITY_HIGH;
    L_Last_First_Fault_Source := GVL_SYSTEM_HEALTH.G_First_Fault_Source;

ELSIF GVL_STATUS.G_Current_Scenario <> GVL_STATUS.G_Previous_Scenario THEN
    L_History_Write_Event := TRUE;
    L_History_Event.event_code := 1001;
    L_History_Event.event_value := TO_REAL(GVL_STATUS.G_Current_Scenario);
    L_History_Event.unit := 4;
    L_History_Event.zone_id := 0;
    L_History_Event.priority := E_ALERT_PRIORITY.ALERT_PRIORITY_HIGH;
    GVL_STATUS.G_Previous_Scenario := GVL_STATUS.G_Current_Scenario;

ELSIF GVL_STATUS.G_Diagnostics.Alarm_Event_Pulse THEN
    L_History_Write_Event := TRUE;
    L_History_Event.event_code := TO_WORD(GVL_STATUS.G_Diagnostics.Alarm_Event_Code);
    L_History_Event.event_value := GVL_STATUS.G_Diagnostics.Alarm_Event_Value;
    L_History_Event.unit := 10;
    L_History_Event.zone_id := 0;
    L_History_Event.priority := E_ALERT_PRIORITY.ALERT_PRIORITY_HIGH;

ELSIF GVL_STATUS.G_Diagnostics.Operator_Journal_Event_Seq <> L_Last_Operator_Journal_Seq THEN
    L_History_Write_Event := TRUE;
    L_History_Event.event_code := 1301;
    L_History_Event.event_value := TO_REAL(GVL_STATUS.G_Diagnostics.Operator_Journal_Event_Seq);
    L_History_Event.unit := 20;
    L_History_Event.zone_id := 0;
    L_History_Event.priority := E_ALERT_PRIORITY.ALERT_PRIORITY_HIGH;
    L_Last_Operator_Journal_Seq := GVL_STATUS.G_Diagnostics.Operator_Journal_Event_Seq;
END_IF;

IF NOT GVL_SYSTEM_HEALTH.G_First_Fault_Active THEN
    L_Last_Root_Cause := GVL_SYSTEM_HEALTH.G_Root_Cause;
    L_Last_First_Fault_Source := GVL_SYSTEM_HEALTH.G_First_Fault_Source;
END_IF;

IF L_History_Write_Event THEN
    IF (L_History_Event.event_code = L_Last_Event_Code)
       AND (ABS(L_History_Event.event_value - L_Last_Event_Value) < 0.001)
       AND (GVL_TIME_SERVICE.G_Now_MS - L_Last_Event_Time_MS < 5000) THEN
        L_History_Write_Event := FALSE;
    ELSE
        L_Last_Event_Code := L_History_Event.event_code;
        L_Last_Event_Value := L_History_Event.event_value;
        L_Last_Event_Time_MS := GVL_TIME_SERVICE.G_Now_MS;
    END_IF;
END_IF;

fbHistoryManager(
    VI_System_Time_MS := GVL_TIME_SERVICE.G_Now_MS,
    VI_Write_Event := L_History_Write_Event,
    VI_Event := L_History_Event
);

END_PROGRAM

(* ---- PRG_System_Runtime_Base.st ---- *)
PROGRAM PRG_System_Runtime_Base
VAR
    fbSystemInit : FB_System_Init;
    fbSystemRecovery : FB_System_Recovery;
    fbSystemPersist : FB_System_Persist_Manager;

    L_Local_State : ST_System_State_Snapshot;
    L_Remote_State : ST_System_State_Snapshot;

    L_Persist_Buffer : ARRAY[0..4] OF BYTE;
    L_Last_Written_Persist_Buffer : ARRAY[0..4] OF BYTE;
    L_Persist_Buffer_Changed : BOOL;
    L_Last_Persist_Write_MS : UDINT;
    L_Recovery_Done : BOOL;
    L_NVRAM_Cmd : BYTE;
    L_NVRAM_Offset : UDINT;
    L_NVRAM_Done : BOOL;
    L_NVRAM_Err : BOOL;
    L_NVRAM_ErrID : UDINT;
END_VAR

// ======================================================
// SYSTEM RUNTIME BASE
// ======================================================
// Initializes and maintains base system runtime helpers.
//
// Legacy direct-state redundancy orchestration is intentionally
// disconnected from active runtime execution.
// Current HA/distributed runtime path is:
// PRG_Peer_Heartbeat_Ingestion -> PRG_Peer_Session_Publication
// -> PRG_HA_Session_Replication -> distributed ingestion/governors.
//
// Do not reconnect FB_System_Redundancy_Orchestrator here without
// explicit barrier/governance review.
// ======================================================

fbSystemInit(
    VIO_Local_State := L_Local_State,
    VIO_Remote_State := L_Remote_State
);

fbSystemRecovery(
    VIO_Recovery_Done := L_Recovery_Done
);

fbSystemPersist(
    VI_System_Time_MS := GVL_TIME_SERVICE.G_Now_MS,
    VI_IsActivePLC := GVL_STATUS.G_Is_Active_PLC,
    VIO_Persist_Buffer := L_Persist_Buffer,
    VIO_Last_Written_Persist_Buffer := L_Last_Written_Persist_Buffer,
    VIO_Persist_Buffer_Changed := L_Persist_Buffer_Changed,
    VIO_Last_Persist_Write_MS := L_Last_Persist_Write_MS,
    VIO_NVRAM_Cmd := L_NVRAM_Cmd,
    VIO_NVRAM_Offset := L_NVRAM_Offset,
    VIO_NVRAM_Done := L_NVRAM_Done,
    VIO_NVRAM_Err := L_NVRAM_Err,
    VIO_NVRAM_ErrID := L_NVRAM_ErrID
);

// >>> BULK_SYNC_ANCHOR: PRG_System_Runtime_Base <<<
END_PROGRAM

(* ---- PRG_System_Simulation.st ---- *)
PROGRAM PRG_System_Simulation
VAR
    fbSimulation : FB_Simulation_Manager;
    fbPlayback : FB_Presence_Playback;
    L_Playback_Lights : ARRAY[1..32] OF BOOL;
    L_Scenario_Config : ST_Scenario_Config;
    L_Scenario_Index : INT;
END_VAR

GVL_SIMULATION.G_Sim_Heating_Sensor_Fault := FALSE;
GVL_SIMULATION.G_Sim_IO_Fault := FALSE;
GVL_SIMULATION.G_Sim_Low_Pressure := FALSE;
GVL_SIMULATION.G_Sim_Predictive_Pump_Fault := FALSE;
GVL_SIMULATION.G_Sim_Gas_Alarm := FALSE;
GVL_SIMULATION.G_Sim_Leak_Alarm := FALSE;
GVL_SIMULATION.G_Sim_Smoke_Alarm := FALSE;
GVL_SIMULATION.G_Sim_Dual_PLC_Active := FALSE;

IF NOT GVL_SIMULATION.G_Simulation_Enable THEN
    GVL_SIMULATION.G_Test_Running := FALSE;
    GVL_SIMULATION.G_Test_Scenario_Active := FALSE;
    GVL_SIMULATION.G_Test_Expected_Result_Code := 0;
    RETURN;
END_IF;

L_Scenario_Index := TO_INT(GVL_STATUS.G_Current_Scenario);
IF (L_Scenario_Index < 1) OR (L_Scenario_Index > GVL_CONSTANTS.C_MAX_SCENARIOS) THEN
    L_Scenario_Index := 1;
END_IF;
L_Scenario_Config := GVL_CONFIG.G_HMI_Scenario_Configs[L_Scenario_Index];

fbSimulation(
    VI_System_Time_MS := GVL_TIME_SERVICE.G_Now_MS,
    VI_IsActivePLC := GVL_STATUS.G_Is_Active_PLC,
    VI_Scenario := GVL_STATUS.G_Current_Scenario,
    VI_Config := L_Scenario_Config
);

fbPlayback(
    VI_Mode_Record := FALSE,
    VI_Time_Index := GVL_TIME_SERVICE.G_Now_MS,
    VI_Light_Inputs := L_Playback_Lights
);

IF GVL_SIMULATION.G_Test_Start THEN
    GVL_SIMULATION.G_Test_Scenario_Active := TRUE;
    GVL_SIMULATION.G_Test_Started_MS := GVL_TIME_SERVICE.G_Now_MS;
END_IF;

IF GVL_SIMULATION.G_Test_Stop THEN
    GVL_SIMULATION.G_Test_Scenario_Active := FALSE;
END_IF;

GVL_SIMULATION.G_Test_Running := GVL_SIMULATION.G_Test_Scenario_Active;

IF NOT GVL_SIMULATION.G_Test_Scenario_Active THEN
    GVL_SIMULATION.G_Test_Expected_Result_Code := 0;
    RETURN;
END_IF;

CASE GVL_SIMULATION.G_Test_Scenario_ID OF

    0:
        GVL_SIMULATION.G_Sim_Heating_Sensor_Fault := GVL_SIMULATION.G_Inject_Heating_Sensor_Fault;
        GVL_SIMULATION.G_Sim_IO_Fault := GVL_SIMULATION.G_Inject_IO_Fault;
        GVL_SIMULATION.G_Sim_Low_Pressure := GVL_SIMULATION.G_Inject_Low_Pressure;
        GVL_SIMULATION.G_Sim_Predictive_Pump_Fault := GVL_SIMULATION.G_Inject_Predictive_Pump_Fault;
        GVL_SIMULATION.G_Sim_Gas_Alarm := GVL_SIMULATION.G_Inject_Gas_Alarm;
        GVL_SIMULATION.G_Sim_Leak_Alarm := GVL_SIMULATION.G_Inject_Leak_Alarm;
        GVL_SIMULATION.G_Sim_Smoke_Alarm := GVL_SIMULATION.G_Inject_Smoke_Alarm;
        GVL_SIMULATION.G_Sim_Dual_PLC_Active := GVL_SIMULATION.G_Inject_Dual_PLC_Active;
        GVL_SIMULATION.G_Test_Expected_Result_Code := 0;

    1:
        GVL_SIMULATION.G_Sim_Gas_Alarm := TRUE;
        GVL_SIMULATION.G_Test_Expected_Result_Code := 1;

    2:
        GVL_SIMULATION.G_Sim_Leak_Alarm := TRUE;
        GVL_SIMULATION.G_Sim_Low_Pressure := TRUE;
        GVL_SIMULATION.G_Test_Expected_Result_Code := 2;

    3:
        GVL_SIMULATION.G_Sim_Heating_Sensor_Fault := TRUE;
        GVL_SIMULATION.G_Sim_Predictive_Pump_Fault := TRUE;
        GVL_SIMULATION.G_Test_Expected_Result_Code := 2;

    4:
        GVL_SIMULATION.G_Sim_Dual_PLC_Active := TRUE;
        GVL_SIMULATION.G_Test_Expected_Result_Code := 3;

    5:
        GVL_SIMULATION.G_Sim_Gas_Alarm := TRUE;
        GVL_SIMULATION.G_Sim_Leak_Alarm := TRUE;
        GVL_SIMULATION.G_Sim_Smoke_Alarm := TRUE;
        GVL_SIMULATION.G_Sim_Low_Pressure := TRUE;
        GVL_SIMULATION.G_Sim_Predictive_Pump_Fault := TRUE;
        GVL_SIMULATION.G_Test_Expected_Result_Code := 4;

ELSE
        GVL_SIMULATION.G_Test_Expected_Result_Code := 0;
END_CASE;

IF (GVL_TIME_SERVICE.G_Now_MS - GVL_SIMULATION.G_Test_Started_MS) > GVL_SIMULATION.G_Test_Duration_MS THEN
    GVL_SIMULATION.G_Test_Scenario_Active := FALSE;
    GVL_SIMULATION.G_Test_Running := FALSE;
END_IF;

END_PROGRAM
// >>> BULK_SYNC_ANCHOR: PRG_System_Simulation <<<

(* ---- PRG_Temporal_Causality_Closure_Governor.st ---- *)
PROGRAM PRG_Temporal_Causality_Closure_Governor
IF GVL_DISTRIBUTED_SAFETY_REALITY_CONSENSUS_FABRIC.Distributed_Safety_Reality_Consensus_Granted
AND NOT GVL_TEMPORAL_CAUSALITY_CLOSURE_FABRIC.Temporal_Fork_Detected
AND NOT GVL_TEMPORAL_CAUSALITY_CLOSURE_FABRIC.Stale_Causality_Application_Detected
AND NOT GVL_TEMPORAL_CAUSALITY_CLOSURE_FABRIC.Recovery_Before_Revocation_Detected
AND NOT GVL_TEMPORAL_CAUSALITY_CLOSURE_FABRIC.Distributed_Timeline_Drift_Detected THEN

    GVL_TEMPORAL_CAUSALITY_CLOSURE_FABRIC.Temporal_Causality_Closure_Valid := TRUE;
    GVL_TEMPORAL_CAUSALITY_CLOSURE_FABRIC.Temporal_Causality_Closure_Granted := TRUE;
    GVL_TEMPORAL_CAUSALITY_CLOSURE_FABRIC.Temporal_Causality_Coherent := TRUE;
    GVL_TEMPORAL_CAUSALITY_CLOSURE_FABRIC.Monotonic_Reality_Timeline_Valid := TRUE;
    GVL_TEMPORAL_CAUSALITY_CLOSURE_FABRIC.Recovery_Revocation_Ordering_Valid := TRUE;
END_IF;
END_PROGRAM

(* ---- PRG_Temporal_Stability_Governor.st ---- *)
PROGRAM PRG_Temporal_Stability_Governor
VAR
    L_Now_MS : UDINT;
    L_Stability_Valid : BOOL := TRUE;
    L_Error_Code : UDINT := 0;
    L_Error_Text : STRING(160) := '';
END_VAR

L_Now_MS := GVL_STATUS.G_System_Time_MS;
L_Stability_Valid := TRUE;
L_Error_Code := 0;
L_Error_Text := '';

// Fail-safe defaults.
GVL_TEMPORAL_STABILITY.Temporal_Stability_Valid := FALSE;
GVL_TEMPORAL_STABILITY.Temporal_Stability_Granted := FALSE;
GVL_TEMPORAL_STABILITY.Temporal_Stability_Quarantine_Active := TRUE;

GVL_TEMPORAL_STABILITY.Post_Convergence_Stable := FALSE;
GVL_TEMPORAL_STABILITY.No_Oscillation_Detected := FALSE;
GVL_TEMPORAL_STABILITY.No_Relay_Chatter_Detected := FALSE;
GVL_TEMPORAL_STABILITY.Thermal_Slope_Stable := FALSE;
GVL_TEMPORAL_STABILITY.Pressure_Stable := FALSE;
GVL_TEMPORAL_STABILITY.Flow_Stable := FALSE;

// Temporal stability requires completed physical transaction.
IF NOT GVL_PHYSICAL_TRANSACTION.Physical_Transaction_Granted THEN
    L_Stability_Valid := FALSE;
    L_Error_Code := 28000;
    L_Error_Text := 'Physical transaction not granted';
END_IF;

// Start deterministic observation window.
IF L_Stability_Valid
AND NOT GVL_TEMPORAL_STABILITY.Stability_Observation_Window_Active THEN
    GVL_TEMPORAL_STABILITY.Stability_Observation_Window_Active := TRUE;
    GVL_TEMPORAL_STABILITY.Stability_Window_Start_MS := L_Now_MS;
END_IF;

IF GVL_TEMPORAL_STABILITY.Stability_Observation_Window_Active THEN
    GVL_TEMPORAL_STABILITY.Stability_Window_Elapsed_MS :=
        L_Now_MS - GVL_TEMPORAL_STABILITY.Stability_Window_Start_MS;
END_IF;

// Observation window must fully elapse.
IF L_Stability_Valid
AND (GVL_TEMPORAL_STABILITY.Stability_Window_Elapsed_MS <
     GVL_TEMPORAL_STABILITY.Stability_Window_Target_MS) THEN

    L_Stability_Valid := FALSE;
    L_Error_Code := 28001;
    L_Error_Text := 'Temporal observation window not elapsed';
END_IF;

// Delayed instability detection.
IF GVL_TEMPORAL_STABILITY.Post_Convergence_Oscillation_Detected THEN
    L_Stability_Valid := FALSE;
    L_Error_Code := 28002;
    L_Error_Text := 'Post-convergence oscillation detected';
END_IF;

IF GVL_TEMPORAL_STABILITY.Thermal_Inertia_Rebound_Detected THEN
    L_Stability_Valid := FALSE;
    L_Error_Code := 28003;
    L_Error_Text := 'Thermal inertia rebound detected';
END_IF;

IF GVL_TEMPORAL_STABILITY.Pressure_Rebound_Detected THEN
    L_Stability_Valid := FALSE;
    L_Error_Code := 28004;
    L_Error_Text := 'Pressure rebound detected';
END_IF;

IF GVL_TEMPORAL_STABILITY.Relay_Chatter_Detected THEN
    L_Stability_Valid := FALSE;
    L_Error_Code := 28005;
    L_Error_Text := 'Relay chatter detected';
END_IF;

IF GVL_TEMPORAL_STABILITY.Pump_Cavitation_Recovery_Detected THEN
    L_Stability_Valid := FALSE;
    L_Error_Code := 28006;
    L_Error_Text := 'Pump cavitation recovery detected';
END_IF;

IF GVL_TEMPORAL_STABILITY.Delayed_Actuator_Divergence_Detected THEN
    L_Stability_Valid := FALSE;
    L_Error_Code := 28007;
    L_Error_Text := 'Delayed actuator divergence detected';
END_IF;

// Stable physical conditions required.
IF L_Stability_Valid
AND NOT GVL_TEMPORAL_STABILITY.No_Oscillation_Detected THEN
    L_Stability_Valid := FALSE;
    L_Error_Code := 28010;
    L_Error_Text := 'Oscillation-free state not confirmed';
END_IF;

IF L_Stability_Valid
AND NOT GVL_TEMPORAL_STABILITY.No_Relay_Chatter_Detected THEN
    L_Stability_Valid := FALSE;
    L_Error_Code := 28011;
    L_Error_Text := 'Relay chatter-free state not confirmed';
END_IF;

IF L_Stability_Valid
AND NOT GVL_TEMPORAL_STABILITY.Thermal_Slope_Stable THEN
    L_Stability_Valid := FALSE;
    L_Error_Code := 28012;
    L_Error_Text := 'Thermal slope stability missing';
END_IF;

IF L_Stability_Valid
AND NOT GVL_TEMPORAL_STABILITY.Pressure_Stable THEN
    L_Stability_Valid := FALSE;
    L_Error_Code := 28013;
    L_Error_Text := 'Pressure stability missing';
END_IF;

IF L_Stability_Valid
AND NOT GVL_TEMPORAL_STABILITY.Flow_Stable THEN
    L_Stability_Valid := FALSE;
    L_Error_Code := 28014;
    L_Error_Text := 'Flow stability missing';
END_IF;

IF L_Stability_Valid THEN
    GVL_TEMPORAL_STABILITY.Temporal_Stability_Valid := TRUE;
    GVL_TEMPORAL_STABILITY.Temporal_Stability_Granted := TRUE;
    GVL_TEMPORAL_STABILITY.Temporal_Stability_Quarantine_Active := FALSE;

    GVL_TEMPORAL_STABILITY.Post_Convergence_Stable := TRUE;

    GVL_TEMPORAL_STABILITY.Temporal_Stability_Epoch :=
        GVL_PHYSICAL_TRANSACTION.Physical_Transaction_Epoch;

    GVL_TEMPORAL_STABILITY.Temporal_Stability_Epoch_Coherent := TRUE;

    GVL_TEMPORAL_STABILITY.Temporal_Stability_Last_Update_MS :=
        L_Now_MS;

    GVL_TEMPORAL_STABILITY.Temporal_Stability_Lease_Expired := FALSE;

    GVL_TEMPORAL_STABILITY.Temporal_Stability_Last_Error_Code := 0;
    GVL_TEMPORAL_STABILITY.Temporal_Stability_Last_Error_Text := '';
ELSE
    GVL_TEMPORAL_STABILITY.Temporal_Stability_Valid := FALSE;
    GVL_TEMPORAL_STABILITY.Temporal_Stability_Granted := FALSE;
    GVL_TEMPORAL_STABILITY.Temporal_Stability_Quarantine_Active := TRUE;

    GVL_TEMPORAL_STABILITY.Temporal_Stability_Lease_Expired := TRUE;

    GVL_TEMPORAL_STABILITY.Temporal_Stability_Last_Error_Code :=
        L_Error_Code;

    GVL_TEMPORAL_STABILITY.Temporal_Stability_Last_Error_Text :=
        L_Error_Text;

    GVL_TEMPORAL_STABILITY.Temporal_Stability_Invalidation_Count :=
        GVL_TEMPORAL_STABILITY.Temporal_Stability_Invalidation_Count + 1;
END_IF;

END_PROGRAM

(* ---- PRG_Time_Monotonic_Governor.st ---- *)
PROGRAM PRG_Time_Monotonic_Governor
VAR
    L_Now_MS : UDINT;
    L_Delta_MS : UDINT;
    L_Time_Valid : BOOL := TRUE;
    L_Error_Code : UDINT := 0;
    L_Error_Text : STRING(160) := '';
END_VAR

L_Now_MS := GVL_STATUS.G_System_Time_MS;
L_Time_Valid := TRUE;
L_Error_Code := 0;
L_Error_Text := '';

// ======================================================
// MONOTONIC TIME GOVERNOR
// ======================================================
// Creates monotonic time authority semantics.
// Prevents rollback/reboot resurrection.
// ======================================================

// First initialization.
IF NOT GVL_TIME_MONOTONIC.Monotonic_Time_Initialized THEN
    GVL_TIME_MONOTONIC.Monotonic_Time_Initialized := TRUE;
    GVL_TIME_MONOTONIC.Boot_Generation_ID := GVL_TIME_MONOTONIC.Boot_Generation_ID + 1;
    GVL_TIME_MONOTONIC.Startup_Quarantine_Active := TRUE;
    GVL_TIME_MONOTONIC.Startup_Quarantine_Start_MS := L_Now_MS;
    GVL_TIME_MONOTONIC.Last_Monotonic_Time_MS := L_Now_MS;
END_IF;

GVL_TIME_MONOTONIC.Time_Rollback_Detected := FALSE;
GVL_TIME_MONOTONIC.Time_Overflow_Detected := FALSE;
GVL_TIME_MONOTONIC.Retained_Time_Invalid := FALSE;
GVL_TIME_MONOTONIC.Startup_Quarantine_Release_Allowed := FALSE;

// Rollback detection.
IF L_Now_MS < GVL_TIME_MONOTONIC.Last_Monotonic_Time_MS THEN
    L_Time_Valid := FALSE;
    L_Error_Code := 8000;
    L_Error_Text := 'Monotonic rollback detected';

    GVL_TIME_MONOTONIC.Time_Rollback_Detected := TRUE;
    GVL_TIME_MONOTONIC.Retained_Time_Invalid := TRUE;
END_IF;

// Overflow / invalid delta detection.
L_Delta_MS := L_Now_MS - GVL_TIME_MONOTONIC.Last_Monotonic_Time_MS;

IF L_Time_Valid AND (L_Delta_MS > 60000) THEN
    L_Time_Valid := FALSE;
    L_Error_Code := 8001;
    L_Error_Text := 'Monotonic delta overflow';

    GVL_TIME_MONOTONIC.Time_Overflow_Detected := TRUE;
END_IF;

// Startup quarantine governance.
IF GVL_TIME_MONOTONIC.Startup_Quarantine_Active THEN
    IF (L_Now_MS - GVL_TIME_MONOTONIC.Startup_Quarantine_Start_MS) >= GVL_TIME_MONOTONIC.Startup_Quarantine_Timeout_MS THEN
        GVL_TIME_MONOTONIC.Startup_Quarantine_Active := FALSE;
        GVL_TIME_MONOTONIC.Startup_Quarantine_Release_Allowed := TRUE;
    ELSE
        L_Time_Valid := FALSE;

        IF L_Error_Code = 0 THEN
            L_Error_Code := 8002;
            L_Error_Text := 'Startup quarantine active';
        END_IF;
    END_IF;
END_IF;

// Publish monotonic authority state.
IF L_Time_Valid THEN
    GVL_TIME_MONOTONIC.Monotonic_Epoch := GVL_TIME_MONOTONIC.Monotonic_Epoch + 1;
    GVL_TIME_MONOTONIC.Monotonic_Time_Valid := TRUE;
    GVL_TIME_MONOTONIC.Last_Validated_Time_MS := L_Now_MS;
    GVL_TIME_MONOTONIC.Last_Monotonic_Time_MS := L_Now_MS;

    GVL_TIME_MONOTONIC.Monotonic_Last_Error_Code := 0;
    GVL_TIME_MONOTONIC.Monotonic_Last_Error_Text := '';
ELSE
    GVL_TIME_MONOTONIC.Monotonic_Time_Valid := FALSE;
    GVL_TIME_MONOTONIC.Monotonic_Last_Error_Code := L_Error_Code;
    GVL_TIME_MONOTONIC.Monotonic_Last_Error_Text := L_Error_Text;

    GVL_TIME_MONOTONIC.Monotonic_Invalidation_Count := GVL_TIME_MONOTONIC.Monotonic_Invalidation_Count + 1;
END_IF;
END_PROGRAM

(* ---- PRG_Time_Service.st ---- *)
PROGRAM PRG_Time_Service
VAR
    fbTimebase : FB_System_Timebase;
    fbTime : FB_Time_Service;
END_VAR

// Central time update point.
// Must run before PRG_IO_Read and all consumers of GVL_TIME_SERVICE.
fbTimebase();
fbTime();

// Step 4.2 compatibility bridge.
// Legacy consumers of GVL_STATUS.G_System_Time_MS receive the same canonical time.
GVL_STATUS.G_System_Time_MS := GVL_TIME_SERVICE.G_Now_MS;
GVL_STATUS.G_Current_TOD := GVL_TIME_SERVICE.G_Current_TOD;
GVL_STATUS.G_Current_Day := TO_UINT(GVL_TIME_SERVICE.G_Day_Of_Week);

END_PROGRAM

(* ---- PRG_Water.st ---- *)
PROGRAM PRG_Water
VAR
    fbProjection : FB_Water_Output_Projection;
    L_Zone_Enable : ARRAY[1..GVL_CONSTANTS.C_MAX_WATER_ZONES] OF BOOL;
    L_Valve_35_Open : BOOL;
    L_Valve_35_Close : BOOL;
    L_Valve_36_Open : BOOL;
    L_Valve_36_Close : BOOL;
    L_Local_Valve_Open : ARRAY[1..6] OF BOOL;
    L_Local_Valve_Close : ARRAY[1..6] OF BOOL;
    L_i : INT;
    L_Projected_Valve_Group : UINT;
END_VAR

// ==============================================================================
// Water runtime output bridge.
//
// Topology:
// - group 1: riser 1 kitchen, local valves 1(HWS/CW) and 2(HW);
// - group 2: riser 2 master bathroom, local valves 3 and 4;
// - group 3: riser 3 guest bathrooms + laundry, local valves 5 and 6;
// - group 4: common inlet 35(CW) and 36(HW).
//
// Normally-open valves are used because water is from a well: no electrical
// power means no pump and no pressurized water. Leak/fallback projects Close;
// HMI emergency-open projects Open for a timed, limited interval.
// ==============================================================================

PRG_Water_Emergency_Open_Manager();

GVL_WATER_DOMAIN_STATUS.G_Runtime_Required := FALSE;
GVL_WATER_DOMAIN_STATUS.G_Runtime_Executed := TRUE;
GVL_WATER_DOMAIN_STATUS.G_Runtime_Idle_By_Design := FALSE;
GVL_WATER_DOMAIN_STATUS.G_Recovery_Requested := FALSE;
GVL_WATER_DOMAIN_STATUS.G_Global_Path_Active := FALSE;
GVL_WATER_DOMAIN_STATUS.G_Output_35_Active := FALSE;
GVL_WATER_DOMAIN_STATUS.G_Output_36_Active := FALSE;
GVL_WATER_DOMAIN_STATUS.G_Any_Zone_Active := FALSE;
GVL_WATER_DOMAIN_STATUS.G_Last_Update_MS := GVL_STATUS.G_System_Time_MS;

FOR L_i := 1 TO GVL_CONSTANTS.C_MAX_WATER_ZONES DO
    L_Zone_Enable[L_i] := FALSE;
END_FOR;

FOR L_i := 1 TO 6 DO
    L_Local_Valve_Open[L_i] := FALSE;
    L_Local_Valve_Close[L_i] := FALSE;
END_FOR;

L_Valve_35_Open := FALSE;
L_Valve_35_Close := FALSE;
L_Valve_36_Open := FALSE;
L_Valve_36_Close := FALSE;

IF GVL_INTENT_SAFETY.I_Water_Selective_Recovery_Allowed THEN
    GVL_WATER_DOMAIN_STATUS.G_Recovery_Requested := TRUE;

    IF (GVL_INTENT_SAFETY.I_Water_Recovery_Target_Zone >= 1) AND (GVL_INTENT_SAFETY.I_Water_Recovery_Target_Zone <= GVL_CONSTANTS.C_MAX_WATER_ZONES) THEN
        L_Zone_Enable[GVL_INTENT_SAFETY.I_Water_Recovery_Target_Zone] := TRUE;
    END_IF;
END_IF;

// Existing authoritative common inlet fallback path from command shadow.
L_Valve_35_Close := GVL_COMMAND_SHADOW.G_Close_Valve_35;
L_Valve_36_Close := GVL_COMMAND_SHADOW.G_Close_Valve_36;

// Deterministic water output projection by isolation group.
IF GVL_Water_Output_Projection.G_Runtime_Valid THEN

    IF GVL_Water_Output_Projection.G_Global_Fallback_Projecting THEN
        FOR L_i := 1 TO 6 DO
            L_Local_Valve_Close[L_i] := TRUE;
        END_FOR;
        L_Valve_35_Close := TRUE;
        L_Valve_36_Close := TRUE;
        GVL_WATER_DOMAIN_STATUS.G_Global_Path_Active := TRUE;
    ELSE
        FOR L_i := 1 TO GVL_CONSTANTS.C_MAX_FLOOD_SENSORS DO
            IF GVL_Water_Output_Projection.G_Output_Projection_State[L_i].Projection_Allowed AND
               GVL_Water_Output_Projection.G_Output_Projection_State[L_i].Physical_Close_Project THEN

                L_Projected_Valve_Group := GVL_Water_Output_Projection.G_Output_Projection_State[L_i].Valve_Group_Id;

                CASE L_Projected_Valve_Group OF
                    1:
                        L_Local_Valve_Close[1] := TRUE;
                        L_Local_Valve_Close[2] := TRUE;
                    2:
                        L_Local_Valve_Close[3] := TRUE;
                        L_Local_Valve_Close[4] := TRUE;
                    3:
                        L_Local_Valve_Close[5] := TRUE;
                        L_Local_Valve_Close[6] := TRUE;
                    4:
                        L_Valve_35_Close := TRUE;
                        L_Valve_36_Close := TRUE;
                ELSE
                    L_Valve_35_Close := TRUE;
                    L_Valve_36_Close := TRUE;
                    GVL_WATER_DOMAIN_STATUS.G_Global_Path_Active := TRUE;
                END_CASE;
            END_IF;
        END_FOR;
    END_IF;
END_IF;

// Emergency open for selected riser/common inlet: project Open and suppress
// the corresponding Close command for the timed interval.
IF GVL_WATER_EMERGENCY_OPEN.G_Open_Riser_1_Active THEN
    L_Local_Valve_Close[1] := FALSE;
    L_Local_Valve_Close[2] := FALSE;
    L_Local_Valve_Open[1] := TRUE;
    L_Local_Valve_Open[2] := TRUE;
END_IF;

IF GVL_WATER_EMERGENCY_OPEN.G_Open_Riser_2_Active THEN
    L_Local_Valve_Close[3] := FALSE;
    L_Local_Valve_Close[4] := FALSE;
    L_Local_Valve_Open[3] := TRUE;
    L_Local_Valve_Open[4] := TRUE;
END_IF;

IF GVL_WATER_EMERGENCY_OPEN.G_Open_Riser_3_Active THEN
    L_Local_Valve_Close[5] := FALSE;
    L_Local_Valve_Close[6] := FALSE;
    L_Local_Valve_Open[5] := TRUE;
    L_Local_Valve_Open[6] := TRUE;
END_IF;

IF GVL_WATER_EMERGENCY_OPEN.G_Open_Common_Inlet_Active THEN
    L_Valve_35_Close := FALSE;
    L_Valve_36_Close := FALSE;
    L_Valve_35_Open := TRUE;
    L_Valve_36_Open := TRUE;
END_IF;

FOR L_i := 1 TO GVL_CONSTANTS.C_MAX_WATER_ZONES DO
    IF L_Zone_Enable[L_i] THEN
        GVL_WATER_DOMAIN_STATUS.G_Any_Zone_Active := TRUE;
    END_IF;
END_FOR;

GVL_WATER_DOMAIN_STATUS.G_Output_35_Active := L_Valve_35_Close OR L_Valve_35_Open;
GVL_WATER_DOMAIN_STATUS.G_Output_36_Active := L_Valve_36_Close OR L_Valve_36_Open;

FOR L_i := 1 TO 6 DO
    IF L_Local_Valve_Close[L_i] OR L_Local_Valve_Open[L_i] THEN
        GVL_WATER_DOMAIN_STATUS.G_Any_Zone_Active := TRUE;
    END_IF;
END_FOR;

GVL_WATER_DOMAIN_STATUS.G_Runtime_Required :=
    GVL_WATER_DOMAIN_STATUS.G_Recovery_Requested
    OR GVL_WATER_DOMAIN_STATUS.G_Global_Path_Active
    OR GVL_WATER_DOMAIN_STATUS.G_Output_35_Active
    OR GVL_WATER_DOMAIN_STATUS.G_Output_36_Active
    OR GVL_WATER_DOMAIN_STATUS.G_Any_Zone_Active;

GVL_WATER_DOMAIN_STATUS.G_Runtime_Idle_By_Design := NOT GVL_WATER_DOMAIN_STATUS.G_Runtime_Required;

IF GVL_WATER_DOMAIN_STATUS.G_Runtime_Idle_By_Design THEN
    GVL_WATER_DOMAIN_STATUS.G_Status_Code := 0;
    GVL_WATER_DOMAIN_STATUS.G_Status_Text := 'Water domain idle by design';
ELSIF GVL_WATER_DOMAIN_STATUS.G_Global_Path_Active THEN
    GVL_WATER_DOMAIN_STATUS.G_Status_Code := 2;
    GVL_WATER_DOMAIN_STATUS.G_Status_Text := 'Water domain global path active';
ELSIF GVL_WATER_EMERGENCY_OPEN.G_Open_Riser_1_Active OR
      GVL_WATER_EMERGENCY_OPEN.G_Open_Riser_2_Active OR
      GVL_WATER_EMERGENCY_OPEN.G_Open_Riser_3_Active OR
      GVL_WATER_EMERGENCY_OPEN.G_Open_Common_Inlet_Active THEN
    GVL_WATER_DOMAIN_STATUS.G_Status_Code := 3;
    GVL_WATER_DOMAIN_STATUS.G_Status_Text := 'Water emergency open active';
ELSE
    GVL_WATER_DOMAIN_STATUS.G_Status_Code := 1;
    GVL_WATER_DOMAIN_STATUS.G_Status_Text := 'Water domain active';
END_IF;

fbProjection(
    VI_Zone_Enable := L_Zone_Enable,
    VI_Valve_35_Open := L_Valve_35_Open,
    VI_Valve_35_Close := L_Valve_35_Close,
    VI_Valve_36_Open := L_Valve_36_Open,
    VI_Valve_36_Close := L_Valve_36_Close,
    VI_Local_Valve_Open := L_Local_Valve_Open,
    VI_Local_Valve_Close := L_Local_Valve_Close
);

// >>> BULK_SYNC_ANCHOR: PRG_Water <<<
END_PROGRAM

(* ---- PRG_Water_Output_Projection.st ---- *)
PROGRAM PRG_Water_Output_Projection
// ==============================================================================
// WATER OUTPUT PROJECTION — deterministic water output runtime boundary.
// ==============================================================================
// Runtime-critical projection/convergence path is separated from observability.
// No authority ownership or command-shadow writes are introduced here.
// ==============================================================================

PRG_Water_Output_Projection_Phase_01_Runtime();
PRG_Water_Output_Projection_Phase_02_Observability();

// Runtime bridge integrated in PRG_Water.
// This PRG remains the deterministic projection boundary.

END_PROGRAM

(* ---- PRG_Water_Output_Projection_Phase_01_Runtime.st ---- *)
PROGRAM PRG_Water_Output_Projection_Phase_01_Runtime
VAR
    fbWaterOutputProjector : FB_Water_Output_Projector;
    fbWaterOutputReconciliation : FB_Water_Output_Reconciliation;
    fbWaterValveFeedback : FB_Water_Valve_Feedback_Runtime;
    fbWaterPhysicalRuntime : FB_Water_Physical_Runtime;
    fbWaterRuntimeHardening : FB_Water_Runtime_Hardening;
    fbWaterRecoveryRuntime : FB_Water_Recovery_Runtime;
END_VAR

// Critical deterministic water output runtime path.
// Must run every PLC scan while water projection is enabled.

fbWaterOutputProjector(
    VI_Enable := TRUE,
    VI_System_Time_MS := GVL_STATUS.G_System_Time_MS
);

fbWaterOutputReconciliation(
    VI_Enable := TRUE,
    VI_System_Time_MS := GVL_STATUS.G_System_Time_MS
);

fbWaterValveFeedback(
    VI_Enable := TRUE,
    VI_System_Time_MS := GVL_STATUS.G_System_Time_MS
);

fbWaterPhysicalRuntime(
    VI_Enable := TRUE,
    VI_System_Time_MS := GVL_STATUS.G_System_Time_MS
);

fbWaterRuntimeHardening(
    VI_Enable := TRUE,
    VI_System_Time_MS := GVL_STATUS.G_System_Time_MS
);

fbWaterRecoveryRuntime(
    VI_Enable := TRUE,
    VI_System_Time_MS := GVL_STATUS.G_System_Time_MS
);

// >>> BULK_SYNC_ANCHOR: PRG_Water_Output_Projection_Phase_01_Runtime <<<
END_PROGRAM
